(* CoDeSys 2.3.9.48 project: 20170913_WUR_added_Inverter_Control.pro *)
(* Version: 0.9 *)
(* Description: Project Distributie Automatisering *)
(* Libraries: Serial_Interface_01.lib 22.4.13 12:50:14, Util.lib 30.1.13 13:05:12, WagoLib787_01.lib 10.11.14 13:02:32, mod_com.lib 30.1.13 13:05:12, WagoConfigToolLIB.lib 30.1.13 13:05:12, PowerMeasurement_495_02.lib 13.9.17 08:23:51, SysLibTime.lib 30.1.13 13:05:12, WagoLibSHA1.lib 19.8.11 14:53:16, WagoLibMySQL_03.lib 23.7.14 09:13:36, SerComm.lib 30.1.13 13:05:12, SysLibSockets.lib 22.5.14 16:16:32, SysLibFile.lib 30.1.13 13:05:12, SysLibMem.lib 30.1.13 13:05:12, SysLibSem.lib 30.1.13 13:05:12, SysLibRtc.lib 30.1.13 13:05:12, WagoLibEthernet_01.lib 1.4.15 14:24:28, WAGOLIBNTP.lib 19.8.11 14:53:14, Modb_l05.lib 13.5.15 10:30:08, SysLibDir.lib 30.1.13 13:05:12, C:\Program Files\WAGO Software\CODESYS V2.3\Targets\WAGO\Libraries\32_Bit\WAGO_Datalogger_02.lib 5.4.17 15:41:49, Wago_MBCFG_SERIAL_01.lib 1.4.15 14:24:28, Wago_MBCFG_COMMON_01.lib 1.4.15 14:24:28, Standard.lib 20.5.14 08:13:26, Iecsfc.lib 30.1.13 13:05:12, SYSLIBCALLBACK.LIB 30.1.13 13:05:12 *)

(* PLC configuration (modules and I/O channels)
0750-0430 8 DI 24 V DC 3.0ms [Type_1_8_Channels] node 0, in %IB264 out %QB280
  AT %IX132.0 [BOOLOnX_I] Ch_1 Digital input
  AT %IX132.1 [BOOLOnX_I] Ch_2 Digital input
  AT %IX132.2 [BOOLOnX_I] Ch_3 Digital input
  AT %IX132.3 [BOOLOnX_I] Ch_4 Digital input
  AT %IX132.4 [BOOLOnX_I] Ch_5 Digital input
  AT %IX132.5 [BOOLOnX_I] Ch_6 Digital input
  AT %IX132.6 [BOOLOnX_I] Ch_7 Digital input
  AT %IX132.7 [BOOLOnX_I] Ch_8 Digital input
0750-0430 8 DI 24 V DC 3.0ms [Type_1_8_Channels] node 1, in %IB264 out %QB280
  AT %IX132.8 [BOOLOnX_I] Ch_1 Digital input
  AT %IX132.9 [BOOLOnX_I] Ch_2 Digital input
  AT %IX132.10 [BOOLOnX_I] Ch_3 Digital input
  AT %IX132.11 [BOOLOnX_I] Ch_4 Digital input
  AT %IX132.12 [BOOLOnX_I] Ch_5 Digital input
  AT %IX132.13 [BOOLOnX_I] Ch_6 Digital input
  AT %IX132.14 [BOOLOnX_I] Ch_7 Digital input
  AT %IX132.15 [BOOLOnX_I] Ch_8 Digital input
0750-0430 8 DI 24 V DC 3.0ms [Type_1_8_Channels] node 2, in %IB265 out %QB280
  AT %IX133.0 [BOOLOnX_I] Ch_1 Digital input
  AT %IX133.1 [BOOLOnX_I] Ch_2 Digital input
  AT %IX133.2 [BOOLOnX_I] Ch_3 Digital input
  AT %IX133.3 [BOOLOnX_I] Ch_4 Digital input
  AT %IX133.4 [BOOLOnX_I] Ch_5 Digital input
  AT %IX133.5 [BOOLOnX_I] Ch_6 Digital input
  AT %IX133.6 [BOOLOnX_I] Ch_7 Digital input
  AT %IX133.7 [BOOLOnX_I] Ch_8 Digital input
0750-0430 8 DI 24 V DC 3.0ms [Type_1_8_Channels] node 3, in %IB266 out %QB280
  AT %IX133.8 [BOOLOnX_I] Ch_1 Digital input
  AT %IX133.9 [BOOLOnX_I] Ch_2 Digital input
  AT %IX133.10 [BOOLOnX_I] Ch_3 Digital input
  AT %IX133.11 [BOOLOnX_I] Ch_4 Digital input
  AT %IX133.12 [BOOLOnX_I] Ch_5 Digital input
  AT %IX133.13 [BOOLOnX_I] Ch_6 Digital input
  AT %IX133.14 [BOOLOnX_I] Ch_7 Digital input
  AT %IX133.15 [BOOLOnX_I] Ch_8 Digital input
0750-0430 8 DI 24 V DC 3.0ms [Type_1_8_Channels] node 4, in %IB267 out %QB280
  AT %IX134.0 [BOOLOnX_I] Ch_1 Digital input
  AT %IX134.1 [BOOLOnX_I] Ch_2 Digital input
  AT %IX134.2 [BOOLOnX_I] Ch_3 Digital input
  AT %IX134.3 [BOOLOnX_I] Ch_4 Digital input
  AT %IX134.4 [BOOLOnX_I] Ch_5 Digital input
  AT %IX134.5 [BOOLOnX_I] Ch_6 Digital input
  AT %IX134.6 [BOOLOnX_I] Ch_7 Digital input
  AT %IX134.7 [BOOLOnX_I] Ch_8 Digital input
0750-0530 8 DO 24 V DC 0.5A [Type_10_8_Channels] node 5, in %IB268 out %QB280
  AT %QX140.0 [BOOLOnX_Q] Ch_1 Digital output
  AT %QX140.1 [BOOLOnX_Q] Ch_2 Digital output
  AT %QX140.2 [BOOLOnX_Q] Ch_3 Digital output
  AT %QX140.3 [BOOLOnX_Q] Ch_4 Digital output
  AT %QX140.4 [BOOLOnX_Q] Ch_5 Digital output
  AT %QX140.5 [BOOLOnX_Q] Ch_6 Digital output
  AT %QX140.6 [BOOLOnX_Q] Ch_7 Digital output
  AT %QX140.7 [BOOLOnX_Q] Ch_8 Digital output
0750-0530 8 DO 24 V DC 0.5A [Type_10_8_Channels] node 6, in %IB269 out %QB280
  AT %QX140.8 [BOOLOnX_Q] Ch_1 Digital output
  AT %QX140.9 [BOOLOnX_Q] Ch_2 Digital output
  AT %QX140.10 [BOOLOnX_Q] Ch_3 Digital output
  AT %QX140.11 [BOOLOnX_Q] Ch_4 Digital output
  AT %QX140.12 [BOOLOnX_Q] Ch_5 Digital output
  AT %QX140.13 [BOOLOnX_Q] Ch_6 Digital output
  AT %QX140.14 [BOOLOnX_Q] Ch_7 Digital output
  AT %QX140.15 [BOOLOnX_Q] Ch_8 Digital output
0750-0530 8 DO 24 V DC 0.5A [Type_10_8_Channels] node 7, in %IB269 out %QB281
  AT %QX141.0 [BOOLOnX_Q] Ch_1 Digital output
  AT %QX141.1 [BOOLOnX_Q] Ch_2 Digital output
  AT %QX141.2 [BOOLOnX_Q] Ch_3 Digital output
  AT %QX141.3 [BOOLOnX_Q] Ch_4 Digital output
  AT %QX141.4 [BOOLOnX_Q] Ch_5 Digital output
  AT %QX141.5 [BOOLOnX_Q] Ch_6 Digital output
  AT %QX141.6 [BOOLOnX_Q] Ch_7 Digital output
  AT %QX141.7 [BOOLOnX_Q] Ch_8 Digital output
0750-0530 8 DO 24 V DC 0.5A [Type_10_8_Channels] node 8, in %IB269 out %QB282
  AT %QX141.8 [BOOLOnX_Q] Ch_1 Digital output
  AT %QX141.9 [BOOLOnX_Q] Ch_2 Digital output
  AT %QX141.10 [BOOLOnX_Q] Ch_3 Digital output
  AT %QX141.11 [BOOLOnX_Q] Ch_4 Digital output
  AT %QX141.12 [BOOLOnX_Q] Ch_5 Digital output
  AT %QX141.13 [BOOLOnX_Q] Ch_6 Digital output
  AT %QX141.14 [BOOLOnX_Q] Ch_7 Digital output
  AT %QX141.15 [BOOLOnX_Q] Ch_8 Digital output
AT %QW0 [WORDOnW_Q] Ch_1 Analog output
AT %QW1 [WORDOnW_Q] Ch_2 Analog output
AT %QW2 [WORDOnW_Q] Ch_3 Analog output
AT %QW3 [WORDOnW_Q] Ch_4 Analog output
AT %QW4 [WORDOnW_Q] Ch_1 Analog output
AT %QW5 [WORDOnW_Q] Ch_2 Analog output
AT %QW6 [WORDOnW_Q] Ch_3 Analog output
AT %QW7 [WORDOnW_Q] Ch_4 Analog output
0750-0495/0000-0001 3-phase PoM690/ 5A [Type_58_1_Channels] node 11, in %IB240 out %QB264
  AT %IW0 [WORDOnW_I] Status Word
  AT %IW1 [WORDOnW_I] Status Word 1
  AT %IW2 [WORDOnW_I] Status Word 2
  AT %IW3 [WORDOnW_I] Status Word 3
  AT %ID2 [DWORDOnD_I] process value 1
  AT %ID3 [DWORDOnD_I] process value 2
  AT %ID4 [DWORDOnD_I] process value 3
  AT %ID5 [DWORDOnD_I] process value 4
  AT %QW8 [WORDOnW_Q] Control Word
  AT %QW9 [WORDOnW_Q] Control Word 1
  AT %QW10 [WORDOnW_Q] Control Word 2
  AT %QW11 [WORDOnW_Q] Control Word 3
0750-0495/0000-0001 3-phase PoM690/ 5A [Type_58_1_Channels] node 12, in %IB240 out %QB272
  AT %IW12 [WORDOnW_I] Status Word
  AT %IW13 [WORDOnW_I] Status Word 1
  AT %IW14 [WORDOnW_I] Status Word 2
  AT %IW15 [WORDOnW_I] Status Word 3
  AT %ID8 [DWORDOnD_I] process value 1
  AT %ID9 [DWORDOnD_I] process value 2
  AT %ID10 [DWORDOnD_I] process value 3
  AT %ID11 [DWORDOnD_I] process value 4
  AT %QW20 [WORDOnW_Q] Control Word
  AT %QW21 [WORDOnW_Q] Control Word 1
  AT %QW22 [WORDOnW_Q] Control Word 2
  AT %QW23 [WORDOnW_Q] Control Word 3
0750-0495/0000-0001 3-phase PoM690/ 5A [Type_58_1_Channels] node 13, in %IB264 out %QB296
  AT %IW24 [WORDOnW_I] Status Word
  AT %IW25 [WORDOnW_I] Status Word 1
  AT %IW26 [WORDOnW_I] Status Word 2
  AT %IW27 [WORDOnW_I] Status Word 3
  AT %ID14 [DWORDOnD_I] process value 1
  AT %ID15 [DWORDOnD_I] process value 2
  AT %ID16 [DWORDOnD_I] process value 3
  AT %ID17 [DWORDOnD_I] process value 4
  AT %QW32 [WORDOnW_Q] Control Word
  AT %QW33 [WORDOnW_Q] Control Word 1
  AT %QW34 [WORDOnW_Q] Control Word 2
  AT %QW35 [WORDOnW_Q] Control Word 3
0750-0495/0000-0001 3-phase PoM690/ 5A [Type_58_1_Channels] node 14, in %IB288 out %QB320
  AT %IW36 [WORDOnW_I] Status Word
  AT %IW37 [WORDOnW_I] Status Word 1
  AT %IW38 [WORDOnW_I] Status Word 2
  AT %IW39 [WORDOnW_I] Status Word 3
  AT %ID20 [DWORDOnD_I] process value 1
  AT %ID21 [DWORDOnD_I] process value 2
  AT %ID22 [DWORDOnD_I] process value 3
  AT %ID23 [DWORDOnD_I] process value 4
  AT %QW44 [WORDOnW_Q] Control Word
  AT %QW45 [WORDOnW_Q] Control Word 1
  AT %QW46 [WORDOnW_Q] Control Word 2
  AT %QW47 [WORDOnW_Q] Control Word 3
0750-0495/0000-0001 3-phase PoM690/ 5A [Type_58_1_Channels] node 15, in %IB312 out %QB344
  AT %IW48 [WORDOnW_I] Status Word
  AT %IW49 [WORDOnW_I] Status Word 1
  AT %IW50 [WORDOnW_I] Status Word 2
  AT %IW51 [WORDOnW_I] Status Word 3
  AT %ID26 [DWORDOnD_I] process value 1
  AT %ID27 [DWORDOnD_I] process value 2
  AT %ID28 [DWORDOnD_I] process value 3
  AT %ID29 [DWORDOnD_I] process value 4
  AT %QW56 [WORDOnW_Q] Control Word
  AT %QW57 [WORDOnW_Q] Control Word 1
  AT %QW58 [WORDOnW_Q] Control Word 2
  AT %QW59 [WORDOnW_Q] Control Word 3
0750-0495/0000-0001 3-phase PoM690/ 5A [Type_58_1_Channels] node 16, in %IB336 out %QB368
  AT %IW60 [WORDOnW_I] Status Word
  AT %IW61 [WORDOnW_I] Status Word 1
  AT %IW62 [WORDOnW_I] Status Word 2
  AT %IW63 [WORDOnW_I] Status Word 3
  AT %ID32 [DWORDOnD_I] process value 1
  AT %ID33 [DWORDOnD_I] process value 2
  AT %ID34 [DWORDOnD_I] process value 3
  AT %ID35 [DWORDOnD_I] process value 4
  AT %QW68 [WORDOnW_Q] Control Word
  AT %QW69 [WORDOnW_Q] Control Word 1
  AT %QW70 [WORDOnW_Q] Control Word 2
  AT %QW71 [WORDOnW_Q] Control Word 3
0750-0495/0000-0001 3-phase PoM690/ 5A [Type_58_1_Channels] node 17, in %IB360 out %QB392
  AT %IW72 [WORDOnW_I] Status Word
  AT %IW73 [WORDOnW_I] Status Word 1
  AT %IW74 [WORDOnW_I] Status Word 2
  AT %IW75 [WORDOnW_I] Status Word 3
  AT %ID38 [DWORDOnD_I] process value 1
  AT %ID39 [DWORDOnD_I] process value 2
  AT %ID40 [DWORDOnD_I] process value 3
  AT %ID41 [DWORDOnD_I] process value 4
  AT %QW80 [WORDOnW_Q] Control Word
  AT %QW81 [WORDOnW_Q] Control Word 1
  AT %QW82 [WORDOnW_Q] Control Word 2
  AT %QW83 [WORDOnW_Q] Control Word 3
0750-0495/0000-0001 3-phase PoM690/ 5A [Type_58_1_Channels] node 18, in %IB384 out %QB416
  AT %IW84 [WORDOnW_I] Status Word
  AT %IW85 [WORDOnW_I] Status Word 1
  AT %IW86 [WORDOnW_I] Status Word 2
  AT %IW87 [WORDOnW_I] Status Word 3
  AT %ID44 [DWORDOnD_I] process value 1
  AT %ID45 [DWORDOnD_I] process value 2
  AT %ID46 [DWORDOnD_I] process value 3
  AT %ID47 [DWORDOnD_I] process value 4
  AT %QW92 [WORDOnW_Q] Control Word
  AT %QW93 [WORDOnW_Q] Control Word 1
  AT %QW94 [WORDOnW_Q] Control Word 2
  AT %QW95 [WORDOnW_Q] Control Word 3
0750-0495/0000-0001 3-phase PoM690/ 5A [Type_58_1_Channels] node 19, in %IB408 out %QB440
  AT %IW96 [WORDOnW_I] Status Word
  AT %IW97 [WORDOnW_I] Status Word 1
  AT %IW98 [WORDOnW_I] Status Word 2
  AT %IW99 [WORDOnW_I] Status Word 3
  AT %ID50 [DWORDOnD_I] process value 1
  AT %ID51 [DWORDOnD_I] process value 2
  AT %ID52 [DWORDOnD_I] process value 3
  AT %ID53 [DWORDOnD_I] process value 4
  AT %QW104 [WORDOnW_Q] Control Word
  AT %QW105 [WORDOnW_Q] Control Word 1
  AT %QW106 [WORDOnW_Q] Control Word 2
  AT %QW107 [WORDOnW_Q] Control Word 3
0750-0495/0000-0001 3-phase PoM690/ 5A [Type_58_1_Channels] node 20, in %IB432 out %QB464
  AT %IW108 [WORDOnW_I] Status Word
  AT %IW109 [WORDOnW_I] Status Word 1
  AT %IW110 [WORDOnW_I] Status Word 2
  AT %IW111 [WORDOnW_I] Status Word 3
  AT %ID56 [DWORDOnD_I] process value 1
  AT %ID57 [DWORDOnD_I] process value 2
  AT %ID58 [DWORDOnD_I] process value 3
  AT %ID59 [DWORDOnD_I] process value 4
  AT %QW116 [WORDOnW_Q] Control Word
  AT %QW117 [WORDOnW_Q] Control Word 1
  AT %QW118 [WORDOnW_Q] Control Word 2
  AT %QW119 [WORDOnW_Q] Control Word 3
0750-0495/0000-0001 3-phase PoM690/ 5A [Type_58_1_Channels] node 0, in %IB456 out %QB488
  AT %IW120 [WORDOnW_I] Status Word
  AT %IW121 [WORDOnW_I] Status Word 1
  AT %IW122 [WORDOnW_I] Status Word 2
  AT %IW123 [WORDOnW_I] Status Word 3
  AT %ID62 [DWORDOnD_I] process value 1
  AT %ID63 [DWORDOnD_I] process value 2
  AT %ID64 [DWORDOnD_I] process value 3
  AT %ID65 [DWORDOnD_I] process value 4
  AT %QW128 [WORDOnW_Q] Control Word
  AT %QW129 [WORDOnW_Q] Control Word 1
  AT %QW130 [WORDOnW_Q] Control Word 2
  AT %QW131 [WORDOnW_Q] Control Word 3
REAL, Fieldbus output [MODBUS_REAL_OUT] node 0, in %IB0 out %QB0
  mb_var0 AT %QD500 [REALOnD_Q] TEST
Modbus-Master [MB_MASTER] node 2, in %IB0 out %QB0
*)

(* Task configuration *)
TASK Test (PRIORITY := 2); (* freewheeling *)
	variables_to_system_array();
	SynchroniserSwitch();
	Group2();
END_TASK
TASK WriteData (PRIORITY := 31, INTERVAL := T#1000ms);
	WRITE_DATA();
END_TASK
TASK Switching (PRIORITY := 3); (* freewheeling *)
	Group1();
END_TASK
TASK Measurements (PRIORITY := 1); (* freewheeling *)
	run_PQ();
END_TASK
TASK Control (PRIORITY := 0, INTERVAL := T#1000ms);
	CHP_Controller();
	EV_Controller();
	Mixer_Controller();
	Inverter_Control_1();
	Inverter_Control_2();
END_TASK

(* Global variable list: Global_Variables *)
VAR_GLOBAL
(* testing purpose values *)
	x																:	 REAL:=1;

(* internally used variables *)
	r_Battery_Bus_Frequency									:	 REAL;
	r_Battery_Bus_Voltage										:	 REAL;
	r_Grid_Bus_Frequency										:	 REAL;
	r_Grid_Bus_Voltage											:	 REAL;

(* Array containing all the system parameters. Values are accessable through modbus tcp starting from register 12288. REAL uses two registers per variable *)
	arSystemState									AT %MW0	:	ARRAY[0.. iNumberSystemVar] OF REAL;
	arSystemStateNames										:	ARRAY[0.. iNumberSystemVar] OF STRING; (* names of registers used in mysql write *)

 (*Measurement values for cards*)
	arMeasurementsGroup1							:	ARRAY[1.. iNumberMeasurementVar] OF REAL;
	arMeasurementsGroup2							:	ARRAY[1.. iNumberMeasurementVar] OF REAL;
	arMeasurementsGroup3							:	ARRAY[1.. iNumberMeasurementVar] OF REAL;
	arMeasurementsGroup4							:	ARRAY[1.. iNumberMeasurementVar] OF REAL;
	arMeasurementsGroup5							:	ARRAY[1.. iNumberMeasurementVar] OF REAL;
	arMeasurementsGroup6							:	ARRAY[1.. iNumberMeasurementVar] OF REAL;
	arMeasurementsGroup7							:	ARRAY[1.. iNumberMeasurementVar] OF REAL;
	arMeasurementsGroup8							:	ARRAY[1.. iNumberMeasurementVar] OF REAL;
	arMeasurementsGroup9							:	ARRAY[1.. iNumberMeasurementVar] OF REAL;
	arMeasurementsGroupA							:	ARRAY[1.. iNumberMeasurementVar] OF REAL;
	arMeasurementsGroupB							:	ARRAY[1.. iNumberMeasurementVar] OF REAL;

 (*Measurement values for bus connector from janitza*)
(* ___ OLD____
	r_modbus_Bus_Connector_L1_P				:  REAL;
	r_modbus_Bus_Connector_L2_P				:  REAL;
	r_modbus_Bus_Connector_L3_P				:  REAL;
	r_modbus_Bus_Connector_L1_Q				:  REAL;
	r_modbus_Bus_Connector_L2_Q				:  REAL;
	r_modbus_Bus_Connector_L3_Q				:  REAL;
	r_modbus_Bus_Connector_L1_V				:  REAL;
	r_modbus_Bus_Connector_L2_V				:  REAL;
	r_modbus_Bus_Connector_L3_V				:  REAL;
	r_modbus_Bus_Connector_L1_I				:  REAL;
	r_modbus_Bus_Connector_L2_I				:  REAL;
	r_modbus_Bus_Connector_L3_I				:  REAL;
	r_modbus_Bus_Connector_L1_f				:  REAL;
	r_modbus_Bus_Connector_L2_f				:  REAL;
	r_modbus_Bus_Connector_L3_f				:  REAL;
*)
	Bus_Connector_L1_P : REAL;
	Bus_Connector_L2_P : REAL;
	Bus_Connector_L3_P : REAL;
	Bus_Connector_L1_Q : REAL;
	Bus_Connector_L2_Q : REAL;
	Bus_Connector_L3_Q : REAL;
	Bus_Connector_L1_V : REAL;
	Bus_Connector_L2_V : REAL;
	Bus_Connector_L3_V : REAL;
	Bus_Connector_L1_I : REAL;
	Bus_Connector_L2_I : REAL;
	Bus_Connector_L3_I : REAL;
	Bus_Connector_L1_f : REAL;
	Bus_Connector_L2_f : REAL;
	Bus_Connector_L3_f : REAL;
	Bus_Connector_3F_radians : REAL;

(* DEIF SYNCHRONISER SWITCHING VARIABLES (including variable set from modbus object < doesnt exist jet *)
(* ___OLD ___
	r_modbus_Synchroniser_state					:	REAL:= 1; (* 0 = deny, 1 = allow, 2 = close request*)
	r_modbus_Synchroniser_Denied_Request		:	BOOL;
	r_modbus_Synchroniser_Close_Request		:	BOOL;

	r_DI_Synchroniser_Close_Request				:	BOOL;
	r_DI_Synchroniser_Denied_Request			:	BOOL;
	r_DI_Synchroniser_Closed						:	BOOL;

	r_Synchroniser_Close_Request_Relais		:	BOOL;
	r_Synchroniser_Close_Denied_Relais			:	BOOL; (* only inplemented if hardware output is available (to control panelel LED*)
*)

	Bus_Connector_3F_Sync_close_requested   			AT %QX129.2 : BOOL;
	Bus_Connector_3F_Sync_closed   						AT %IX121.12 : BOOL;
	Bus_Connector_3F_Sync_close_requested_panel    	AT %IX121.13 : BOOL;
	Bus_Connector_3F_Sync_denied_panel   				AT %IX121.14 : BOOL;
	Bus_Connector_3F_Sync_close_requested_modbus 					: BOOL;
	Bus_Connector_3F_Sync_denied_modbus				 				: BOOL;
	Bus_Connector_3F_Field_Rotation										: REAL;
	r_Synchroniser_Close_Denied_Relais (* ?LED? *)						: BOOL;


(* Group Switching states ______ OLD__________
	Group1_autoswitch_state 						(*AT %IX0.0*)	:	BOOL;
	Group1_gridbus_switch_state 					(*AT %QX0.0*)	:	BOOL;
	Group1_batterybus_switch_state 				(*AT %QX0.0*)	:	BOOL;
	Group2_autoswitch_state 						(*AT %IX0.0*)	:	BOOL;
	Group2_gridbus_switch_state 					(*AT %QX0.0*)	:	BOOL;
	Group2_batterybus_switch_state 				(*AT %QX0.0*)	:	BOOL;
	Group3_autoswitch_state 						(*AT %IX0.0*)	:	BOOL;
	Group3_gridbus_switch_state 					(*AT %QX0.0*)	:	BOOL;
	Group3_batterybus_switch_state 				(*AT %QX0.0*)	:	BOOL;
	Group4_autoswitch_state 						(*AT %IX0.0*)	:	BOOL;
	Group4_gridbus_switch_state 					(*AT %QX0.0*)	:	BOOL;
	Group4_batterybus_switch_state 				(*AT %QX0.0*)	:	BOOL;
	Group5_autoswitch_state 						(*AT %IX0.0*)	:	BOOL;
	Group5_gridbus_switch_state 					(*AT %QX0.0*)	:	BOOL;
	Group5_batterybus_switch_state 				(*AT %QX0.0*)	:	BOOL;
	Group6_autoswitch_state 						(*AT %IX0.0*)	:	BOOL;
	Group6_gridbus_switch_state 					(*AT %QX0.0*)	:	BOOL;
	Group6_batterybus_switch_state 				(*AT %QX0.0*)	:	BOOL;
	Group7_autoswitch_state 						(*AT %IX0.0*)	:	BOOL;
	Group7_gridbus_switch_state 					(*AT %QX0.0*)	:	BOOL;
	Group7_batterybus_switch_state 				(*AT %QX0.0*)	:	BOOL;
	Group8_autoswitch_state 						(*AT %IX0.0*)	:	BOOL;
	Group8_gridbus_switch_state 					(*AT %QX0.0*)	:	BOOL;
	Group8_batterybus_switch_state 				(*AT %QX0.0*)	:	BOOL;
	Group9_autoswitch_state 						(*AT %IX0.0*)	:	BOOL;
	Group9_gridbus_switch_state 					(*AT %QX0.0*)	:	BOOL;
	Group9_batterybus_switch_state 				(*AT %QX0.0*)	:	BOOL;
	Group10_autoswitch_state 						(*AT %IX0.0*)	:	BOOL;
	Group10_gridbus_switch_state 					(*AT %QX0.0*)	:	BOOL;
	Group10_batterybus_switch_state 				(*AT %QX0.0*)	:	BOOL;
	Group11_autoswitch_state 						(*AT %IX0.0*)	:	BOOL;
	Group11_gridbus_switch_state 					(*AT %QX0.0*)	:	BOOL;
	Group11_batterybus_switch_state 				(*AT %QX0.0*)	:	BOOL;
*)

	Group_control_Frequencybased_bus_selecting_state : REAL:=0;
	Group_control_min_time_above_switch_frequency : REAL := 2000;
	Group_control_min_time_below_switch_frequency : REAL := 2000;
	Group1_3F_Switch_frequency_to_batterybus : REAL;
	Group1_3F_Switch_frequency_to_gridbus : REAL;
	Group1_3F_min_time_between_switching : REAL:= 10000;
	Group2_3F_Switch_frequency_to_batterybus : REAL := 51;
	Group2_3F_Switch_frequency_to_gridbus : REAL := 49;
	Group2_3F_min_time_between_switching : REAL := 10000;
	Group3_3F_Switch_frequency_to_batterybus : REAL;
	Group3_3F_Switch_frequency_to_gridbus : REAL;
	Group3_3F_min_time_between_switching : REAL;
	Group4_3F_Switch_frequency_to_batterybus : REAL;
	Group4_3F_Switch_frequency_to_gridbus : REAL;
	Group4_3F_min_time_between_switching : REAL;
	Group5_3F_Switch_frequency_to_batterybus : REAL;
	Group5_3F_Switch_frequency_to_gridbus : REAL;
	Group5_3F_min_time_between_switching : REAL;
	Group6_3F_Switch_frequency_to_batterybus : REAL;
	Group6_3F_Switch_frequency_to_gridbus : REAL;
	Group6_3F_min_time_between_switching : REAL;
	Group7_3F_Switch_frequency_to_batterybus : REAL;
	Group7_3F_Switch_frequency_to_gridbus : REAL;
	Group7_3F_min_time_between_switching : REAL;
	Group8_3F_Switch_frequency_to_batterybus : REAL;
	Group8_3F_Switch_frequency_to_gridbus : REAL;
	Group8_3F_min_time_between_switching : REAL;
	Group9_3F_Switch_frequency_to_batterybus : REAL;
	Group9_3F_Switch_frequency_to_gridbus : REAL;
	Group9_3F_min_time_between_switching : REAL;

(* frequency based swithcing parameters *)
	Frequencybased_bus_selecting_state							:  BOOL	:= FALSE;
	Switch_Gap_Time												:  INT		:= 2000;
(*
	Group1_Switch_frequency_to_batterybus						:  REAL	 := 52;
	Group1_Switch_frequency_to_gridbus							:  REAL	 := 48;
	Group1_min_time_above_switch_frequency					:  INT 		:= 10000; (*ms*)
	Group1_min_time_below_switch_frequency					:  INT 		:= 10000; (*ms*)
	Group1_min_time_between_switching							:  INT 		:= 10000; (*ms*)
	Group2_Switch_frequency_to_batterybus						:  REAL 	:= 52;
	Group2_Switch_frequency_to_gridbus							:  REAL 	:= 48;
	Group2_min_time_above_switch_frequency					:  INT 		:= 10000; (*ms*)
	Group2_min_time_below_switch_frequency					:  INT 		:= 10000; (*ms*)
	Group2_min_time_between_switching							:  INT 		:= 10000; (*ms*)
	Group3_Switch_frequency_to_batterybus						:  REAL 	:= 52;
	Group3_Switch_frequency_to_gridbus							:  REAL 	:= 48;
	Group3_min_time_above_switch_frequency					:  INT 		:= 10000; (*ms*)
	Group3_min_time_below_switch_frequency					:  INT 		:= 10000; (*ms*)
	Group3_min_time_between_switching							:  INT 		:= 10000; (*ms*)
	Group4_Switch_frequency_to_batterybus						:  REAL 	:= 52;
	Group4_Switch_frequency_to_gridbus							:  REAL 	:= 48;
	Group4_min_time_above_switch_frequency					:  INT 		:= 10000; (*ms*)
	Group4_min_time_below_switch_frequency					:  INT 		:= 10000; (*ms*)
	Group4_min_time_between_switching							:  INT 		:= 10000; (*ms*)
	Group5_Switch_frequency_to_batterybus						:  REAL 	:= 52;
	Group5_Switch_frequency_to_gridbus							:  REAL 	:= 48;
	Group5_min_time_above_switch_frequency					:  INT 		:= 10000; (*ms*)
	Group5_min_time_below_switch_frequency					:  INT 		:= 10000; (*ms*)
	Group5_min_time_between_switching							:  INT 		:= 10000; (*ms*)
	Group6_Switch_frequency_to_batterybus						:  REAL 	:= 52;
	Group6_Switch_frequency_to_gridbus							:  REAL 	:= 48;
	Group6_min_time_above_switch_frequency					:  INT 		:= 10000; (*ms*)
	Group6_min_time_below_switch_frequency					:  INT 		:= 10000; (*ms*)
	Group6_min_time_between_switching							:  INT 		:= 10000; (*ms*)
	Group7_Switch_frequency_to_batterybus						:  REAL 	:= 52;
	Group7_Switch_frequency_to_gridbus							:  REAL 	:= 48;
	Group7_min_time_above_switch_frequency					:  INT 		:= 10000; (*ms*)
	Group7_min_time_below_switch_frequency					:  INT 		:= 10000; (*ms*)
	Group7_min_time_between_switching							:  INT 		:= 10000; (*ms*)
	Group8_Switch_frequency_to_batterybus						:  REAL 	:= 52;
	Group8_Switch_frequency_to_gridbus							:  REAL 	:= 48;
	Group8_min_time_above_switch_frequency					:  INT 		:= 10000; (*ms*)
	Group8_min_time_below_switch_frequency					:  INT 		:= 10000; (*ms*)
	Group8_min_time_between_switching							:  INT 		:= 10000; (*ms*)
	Group9_Switch_frequency_to_batterybus						:  REAL 	:= 52;
	Group9_Switch_frequency_to_gridbus							:  REAL 	:= 48;
	Group9_min_time_above_switch_frequency					:  INT 		:= 10000; (*ms*)
	Group9_min_time_below_switch_frequency					:  INT 		:= 10000; (*ms*)
	Group9_min_time_between_switching							:  INT 		:= 10000; (*ms*)
*)

	CHP_control_grid_bus_select_controlswitch 							: BOOL;
	CHP_control_baterry_bus_select_controlswitch 						: BOOL;
	CHP_control_auto_bus_select_controlswitch 							: BOOL;
	CHP_control_Offgrid_request    							AT %QX129.4  : BOOL;
	CHP_control_internal_contacter_switch_state  			AT %IX121.15 : BOOL;
	CHP_gridbus_switch_state												: BOOL; (*request from battery bus frequency *)
	CHP_batterybus_switch_state											: BOOL; (*request from battery bus frequency *)

	Inverter_10V_control_Max_Freq_Ref							:  INT		:= 51;  (* Maximum freq possible on the battery bus or te highest freq you want to scale the 0-10V analog output to*)
	Inverter_10V_control_Min_Freq_Ref							:  INT		:= 49;  (* Minimum freq possible on the battery bus or te loweste freq you want to scale the 0-10V analog output to*)
(* Analog Out Controller variables *)

	Mixer_control_control_signal 							AT %QW0 : REAL;   (*0-10V*)
	EV_control_control_signal   								AT %QW2 : REAL;   (*0-10V *)
	CHP_control_Offgrid_Active_Power_control				AT %QW4 : REAL;   (* 4-20ma *)
	Inverter_control1_signal   								AT %QW1 : REAL;	  (*0-10V*)
	Inverter_control2_signal									AT %QW3 : REAL;	  (*0-10V*)
	Group1_3F_Auto_relay_control_battery_bus   	AT %QX128.1  : BOOL;
	Group1_3F_Auto_relay_control_grid_bus   		AT %QX128.0  : BOOL;
	Group1_3F_Selector_auto_bus_select    		AT %IX121.2 : BOOL;
	Group1_3F_relay_state_battery_bus   			AT %IX120.1  : BOOL;
	Group1_3F_relay_state_grid_bus   				AT %IX120.0  : BOOL;
	Group2_3F_Auto_relay_control_battery_bus   	AT %QX128.3  : BOOL;
	Group2_3F_Auto_relay_control_grid_bus   		AT %QX128.2  : BOOL;
	Group2_3F_Selector_auto_bus_select  			AT %IX121.3 : BOOL;
	Group2_3F_relay_state_battery_bus   			AT %IX120.3  : BOOL;
	Group2_3F_relay_state_grid_bus   				AT %IX120.2  : BOOL;
	Group3_3F_Auto_relay_control_battery_bus   	AT %QX128.5  : BOOL;
	Group3_3F_Auto_relay_control_grid_bus   		AT %QX128.4  : BOOL;
	Group3_3F_Selector_auto_bus_select   		AT %IX121.4 : BOOL;
	Group3_3F_relay_state_battery_bus   			AT %IX120.5  : BOOL;
	Group3_3F_relay_state_grid_bus   				AT %IX120.4  : BOOL;
	Group4_3F_Auto_relay_control_battery_bus    	AT %QX128.7  : BOOL;
	Group4_3F_Auto_relay_control_grid_bus    		AT %QX128.6  : BOOL;
	Group4_3F_Selector_auto_bus_select   		AT %IX121.5 : BOOL;
	Group4_3F_relay_state_battery_bus   			AT %IX120.7  : BOOL;
	Group4_3F_relay_state_grid_bus   				AT %IX120.6  : BOOL;
	Group5_3F_Auto_relay_control_battery_bus   	AT %QX128.9  : BOOL;
	Group5_3F_Auto_relay_control_grid_bus   		AT %QX128.8  : BOOL;
	Group5_3F_Selector_auto_bus_select   		AT %IX121.6 : BOOL;
	Group5_3F_relay_state_battery_bus   			AT %IX120.9  : BOOL;
	Group5_3F_relay_state_grid_bus   				AT %IX120.8  : BOOL;
	Group6_3F_Auto_relay_control_battery_bus   	AT %QX128.11  : BOOL;
	Group6_3F_Auto_relay_control_grid_bus   		AT %QX128.10  : BOOL;
	Group6_3F_Selector_auto_bus_select   		AT %IX121.7 : BOOL;
	Group6_3F_relay_state_battery_bus   			AT %IX120.11  : BOOL;
	Group6_3F_relay_state_grid_bus   				AT %IX120.10  : BOOL;
	Group7_3F_Auto_relay_control_battery_bus   	AT %QX128.13  : BOOL;
	Group7_3F_Auto_relay_control_grid_bus   		AT %QX128.12  : BOOL;
	Group7_3F_Selector_auto_bus_select   		AT %IX121.8 : BOOL;
	Group7_3F_relay_state_battery_bus   			AT %IX120.13  : BOOL;
	Group7_3F_relay_state_grid_bus   				AT %IX120.12  : BOOL;
	Group8_3F_Auto_relay_control_battery_bus   	AT %QX128.15  : BOOL;
	Group8_3F_Auto_relay_control_grid_bus   		AT %QX128.14  : BOOL;
	Group8_3F_Selector_auto_bus_select   		AT %IX121.9 : BOOL;
	Group8_3F_relay_state_battery_bus   			AT %IX120.15  : BOOL;
	Group8_3F_relay_state_grid_bus   				AT %IX120.14  : BOOL;
	Group9_3F_Auto_relay_control_battery_bus   	AT %QX129.1  : BOOL;
	Group9_3F_Auto_relay_control_grid_bus   		AT %QX129.0  : BOOL;
	Group9_3F_Selector_auto_bus_select   		AT %IX121.10 : BOOL;
	Group9_3F_relay_state_battery_bus   			AT %IX121.1  : BOOL;
	Group9_3F_relay_state_grid_bus   				AT %IX121.0  : BOOL;

(* Controm panel LEDs *)
	Control_panel_status_warning_led   			AT %QX129.12  : BOOL;
	Control_panel_status_error_led   				AT %QX129.13  : BOOL;
	Control_panel_status_operational_led    		AT %QX129.11  : BOOL;

END_VAR

VAR_GLOBAL CONSTANT

(* Read / write CSV-files *)
	iMaxParams			:	INT:=8;(* Number of Parameters per File *)
	gc_ParameterCount	:	INT:=1;(* Number of Values per Parameter *)
	gc_RawDataSize		:	UINT:=500; (* Raw data size for reading in file ASCII *)
	gcRowExcel			:	INT:=1;

(* meaasurement array length *)
	iNumberMeasurementVar		:	INT := 18;
	iNumberMeasurementGroups	:	 INT:= 11;
(* System array length *)
	iNumberSystemVar			:	INT := 300;

(* MySQL *)
	gcMySql_iSqlLength			:	 INT := 370; 		(* Defines the size in byte of an array element of "asSqlStatement", used by function blocks "MySql_ExecSql" and "MySql_Query"
															to provide an SQL statement as "ARRAY [0..UpperBound] OF STRING(Size)".*)
	raw_SQL_STR_LENGTH		:	 INT := 350;

	gc_MaxBufferSize 	       :INT := 5000; (*number of items to hold in memory*)
	gv_iBuffCounter			:INT := 0; (* counter for  buffer*)
	gv_iBuffPointer			:INT := 0; (* pointer  for  buffer*)
	gv_Buffer					:ARRAY[0..gc_MaxBufferSize] OF ARRAY[0.. iNumberSystemVar] OF REAL; (*In memory buffer of failed message attempts*)


	gc_sHost : STRING := '### your mysql server address here';  (*'application.dyndns.info';*)
	gc_uiPort : UINT := 3306;
	gc_sUser : STRING := '### your mysql server username ';
	gc_sPwd : STRING := '### your mysql password';
	gc_sDB : STRING := '### your MYSQL database';   	(* Optional - Name of database instance to connect to *)
	gc_sTable:STRING := '### your MYSql table' ;

END_VAR

VAR_GLOBAL PERSISTENT RETAIN

	CurrentRatioPQ1						:	WORD := 400;			(* Current transformer ratio, eg 5 A / 400 A *)
	CurrentRatioPQ2						:	WORD := 400;

END_VAR

(* Data type *)
TYPE typCSV :
STRUCT
	sDescription	:STRING;
	Parameter		:ARRAY[1..gc_ParameterCount] OF STRING;
END_STRUCT
END_TYPE

(* POU 05. System State Array/variables_to_system_array, ST *)
PROGRAM variables_to_system_array
VAR
	i: INT;
	j: INT;
	start : INT;
END_VAR
(* https://docs.google.com/spreadsheets/d/1TR7oXGZyEmNnGigmreKdtnpXsz8mxFcoB4b4beNITCA/edit *)

(* loop trough all variable and measurements groups *)
FOR j := 0 TO iNumberMeasurementGroups-1 DO

	start := j*iNumberMeasurementVar;
	FOR i := 1 TO iNumberMeasurementVar-1  DO

		IF i +start <= iNumberMeasurementVar THEN
			arSystemState[i+start] := arMeasurementsGroup1[i];
		END_IF

		IF i +start > iNumberMeasurementVar AND  i +start <= 2*iNumberMeasurementVar THEN
			arSystemState[i+start] := arMeasurementsGroup2[i];
		END_IF

		IF i +start > 2*iNumberMeasurementVar AND  i +start <= 3*iNumberMeasurementVar THEN
			arSystemState[i+start] := arMeasurementsGroup3[i];
		END_IF

		IF i +start > 3*iNumberMeasurementVar AND  i +start <= 4*iNumberMeasurementVar THEN
			arSystemState[i+start] := arMeasurementsGroup4[i];
		END_IF

		IF i +start > 4*iNumberMeasurementVar AND  i +start <= 5*iNumberMeasurementVar THEN
			arSystemState[i+start] := arMeasurementsGroup5[i];
		END_IF

		IF i +start > 5*iNumberMeasurementVar AND  i +start <= 6*iNumberMeasurementVar THEN
			arSystemState[i+start] := arMeasurementsGroup6[i];
		END_IF

		IF i +start > 6*iNumberMeasurementVar AND  i +start <= 7*iNumberMeasurementVar THEN
			arSystemState[i+start] := arMeasurementsGroup7[i];
		END_IF
		IF i +start > 7*iNumberMeasurementVar AND  i +start <= 8*iNumberMeasurementVar THEN
			arSystemState[i+start] := arMeasurementsGroup8[i];
		END_IF

		IF i +start > 8*iNumberMeasurementVar AND  i +start <= 9*iNumberMeasurementVar THEN
			arSystemState[i+start] := arMeasurementsGroup9[i];
		END_IF

		IF i +start > 9*iNumberMeasurementVar AND  i +start <= 10*iNumberMeasurementVar THEN
			arSystemState[i+start] := arMeasurementsGroupA[i];
		END_IF

		IF i +start > 10*iNumberMeasurementVar AND  i +start <= 11*iNumberMeasurementVar THEN
			arSystemState[i+start] := arMeasurementsGroupB[i];
		END_IF

	END_FOR
END_FOR

(* _____ ALWAYS UDPATE (REVERSRE) THE WRITABLE MODBUS PARAMETERS _____

Bus_Connector_3F_Sync_close_requested_modbus 					: BOOL;
Bus_Connector_3F_Sync_denied_modbus				 				: BOOL;
example:
	Bus_Connector_3F_Sync_close_requested_modbus:=REAL_TO_BOOL(arSystemState[219]);
	Bus_Connector_3F_Sync_denied_modbus :=REAL_TO_BOOL(arSystemState[220]);
*)

(* other system variable*)
arSystemState[199] :=Bus_Connector_L1_P;
arSystemState[200] :=Bus_Connector_L2_P;
arSystemState[201] :=Bus_Connector_L3_P;
arSystemState[202] :=Bus_Connector_L1_Q;
arSystemState[203] :=Bus_Connector_L2_Q;
arSystemState[204] :=Bus_Connector_L3_Q;
arSystemState[205] :=Bus_Connector_L1_V;
arSystemState[206] :=Bus_Connector_L2_V;
arSystemState[207] :=Bus_Connector_L3_V;
arSystemState[208] :=Bus_Connector_L1_I;
arSystemState[209] :=Bus_Connector_L2_I;
arSystemState[210] :=Bus_Connector_L3_I;
arSystemState[211] :=Bus_Connector_L1_f;
arSystemState[212] :=Bus_Connector_L2_f;
arSystemState[213] :=Bus_Connector_L3_f;
arSystemState[214] :=Bus_Connector_3F_radians;
arSystemState[215] :=BOOL_TO_REAL(Bus_Connector_3F_Sync_close_requested);
arSystemState[216] :=BOOL_TO_REAL(Bus_Connector_3F_Sync_closed);
arSystemState[217] :=BOOL_TO_REAL(Bus_Connector_3F_Sync_close_requested_panel);
arSystemState[218] :=BOOL_TO_REAL(Bus_Connector_3F_Sync_denied_panel);
Bus_Connector_3F_Sync_close_requested_modbus:=REAL_TO_BOOL(arSystemState[219]);
Bus_Connector_3F_Sync_denied_modbus :=REAL_TO_BOOL(arSystemState[220]);
arSystemState[221] :=Bus_Connector_3F_Field_Rotation;
arSystemState[222] :=BOOL_TO_REAL(CHP_control_grid_bus_select_controlswitch);
arSystemState[223] :=BOOL_TO_REAL(CHP_control_baterry_bus_select_controlswitch);
arSystemState[224] :=BOOL_TO_REAL(CHP_control_auto_bus_select_controlswitch);
arSystemState[225] :=BOOL_TO_REAL(CHP_control_Offgrid_request);
arSystemState[226] :=CHP_control_Offgrid_Active_Power_control;
arSystemState[227] :=BOOL_TO_REAL(CHP_control_internal_contacter_switch_state);
arSystemState[228] :=EV_control_control_signal;
arSystemState[229] :=Mixer_control_control_signal;
arSystemState[230] :=BOOL_TO_REAL(Group1_3F_Auto_relay_control_battery_bus);
arSystemState[231] :=BOOL_TO_REAL(Group1_3F_Auto_relay_control_grid_bus);
arSystemState[232] :=BOOL_TO_REAL(Group1_3F_Selector_auto_bus_select);
arSystemState[233] :=BOOL_TO_REAL(Group1_3F_relay_state_battery_bus);
arSystemState[234] :=BOOL_TO_REAL(Group1_3F_relay_state_grid_bus);
arSystemState[233] :=BOOL_TO_REAL(Group2_3F_Auto_relay_control_battery_bus);
arSystemState[234] :=BOOL_TO_REAL(Group2_3F_Auto_relay_control_grid_bus);
arSystemState[235] :=BOOL_TO_REAL(Group2_3F_Selector_auto_bus_select);
arSystemState[236] :=BOOL_TO_REAL(Group2_3F_relay_state_battery_bus);
arSystemState[237] :=BOOL_TO_REAL(Group2_3F_relay_state_grid_bus);
arSystemState[236] :=BOOL_TO_REAL(Group3_3F_Auto_relay_control_battery_bus);
arSystemState[237] :=BOOL_TO_REAL(Group3_3F_Auto_relay_control_grid_bus);
arSystemState[238] :=BOOL_TO_REAL(Group3_3F_Selector_auto_bus_select);
arSystemState[239] :=BOOL_TO_REAL(Group3_3F_relay_state_battery_bus);
arSystemState[240] :=BOOL_TO_REAL(Group3_3F_relay_state_grid_bus);
arSystemState[239] :=BOOL_TO_REAL(Group4_3F_Auto_relay_control_battery_bus);
arSystemState[240] :=BOOL_TO_REAL(Group4_3F_Auto_relay_control_grid_bus);
arSystemState[241] :=BOOL_TO_REAL(Group4_3F_Selector_auto_bus_select);
arSystemState[242] :=BOOL_TO_REAL(Group4_3F_relay_state_battery_bus);
arSystemState[243] :=BOOL_TO_REAL(Group4_3F_relay_state_grid_bus);
arSystemState[242] :=BOOL_TO_REAL(Group5_3F_Auto_relay_control_battery_bus);
arSystemState[243] :=BOOL_TO_REAL(Group5_3F_Auto_relay_control_grid_bus);
arSystemState[244] :=BOOL_TO_REAL(Group5_3F_Selector_auto_bus_select);
arSystemState[245] :=BOOL_TO_REAL(Group5_3F_relay_state_battery_bus);
arSystemState[246] :=BOOL_TO_REAL(Group5_3F_relay_state_grid_bus);
arSystemState[245] :=BOOL_TO_REAL(Group6_3F_Auto_relay_control_battery_bus);
arSystemState[246] :=BOOL_TO_REAL(Group6_3F_Auto_relay_control_grid_bus);
arSystemState[247] :=BOOL_TO_REAL(Group6_3F_Selector_auto_bus_select);
arSystemState[248] :=BOOL_TO_REAL(Group6_3F_relay_state_battery_bus);
arSystemState[249] :=BOOL_TO_REAL(Group6_3F_relay_state_grid_bus);
arSystemState[248] :=BOOL_TO_REAL(Group7_3F_Auto_relay_control_battery_bus);
arSystemState[249] :=BOOL_TO_REAL(Group7_3F_Auto_relay_control_grid_bus);
arSystemState[250] :=BOOL_TO_REAL(Group7_3F_Selector_auto_bus_select);
arSystemState[251] :=BOOL_TO_REAL(Group7_3F_relay_state_battery_bus);
arSystemState[252] :=BOOL_TO_REAL(Group7_3F_relay_state_grid_bus);
arSystemState[251] :=BOOL_TO_REAL(Group8_3F_Auto_relay_control_battery_bus);
arSystemState[252] :=BOOL_TO_REAL(Group8_3F_Auto_relay_control_grid_bus);
arSystemState[253] :=BOOL_TO_REAL(Group8_3F_Selector_auto_bus_select);
arSystemState[254] :=BOOL_TO_REAL(Group8_3F_relay_state_battery_bus);
arSystemState[255] :=BOOL_TO_REAL(Group8_3F_relay_state_grid_bus);
arSystemState[256] :=BOOL_TO_REAL(Group9_3F_Auto_relay_control_battery_bus);
arSystemState[257] :=BOOL_TO_REAL(Group9_3F_Auto_relay_control_grid_bus);
arSystemState[258] :=BOOL_TO_REAL(Group9_3F_Selector_auto_bus_select);
arSystemState[259] :=BOOL_TO_REAL(Group9_3F_relay_state_battery_bus);
arSystemState[260] :=BOOL_TO_REAL(Group9_3F_relay_state_grid_bus);
arSystemState[261] :=Group_control_Frequencybased_bus_selecting_state;
arSystemState[262] :=Group_control_min_time_above_switch_frequency;
arSystemState[263] :=Group_control_min_time_below_switch_frequency;
arSystemState[264] :=Group1_3F_Switch_frequency_to_batterybus;
arSystemState[265] :=Group1_3F_Switch_frequency_to_gridbus;
arSystemState[266] :=Group1_3F_min_time_between_switching;
arSystemState[267] :=Group2_3F_Switch_frequency_to_batterybus;
arSystemState[268] :=Group2_3F_Switch_frequency_to_gridbus;
arSystemState[269] :=Group2_3F_min_time_between_switching;
arSystemState[268] :=Group3_3F_Switch_frequency_to_batterybus;
arSystemState[269] :=Group3_3F_Switch_frequency_to_gridbus;
arSystemState[270] :=Group3_3F_min_time_between_switching;
arSystemState[271] :=Group4_3F_Switch_frequency_to_batterybus;
arSystemState[270] :=Group4_3F_Switch_frequency_to_gridbus;
arSystemState[271] :=Group4_3F_min_time_between_switching;
arSystemState[272] :=Group5_3F_Switch_frequency_to_batterybus;
arSystemState[273] :=Group5_3F_Switch_frequency_to_gridbus;
arSystemState[272] :=Group5_3F_min_time_between_switching;
arSystemState[273] :=Group6_3F_Switch_frequency_to_batterybus;
arSystemState[274] :=Group6_3F_Switch_frequency_to_gridbus;
arSystemState[275] :=Group6_3F_min_time_between_switching;
arSystemState[274] :=Group7_3F_Switch_frequency_to_batterybus;
arSystemState[275] :=Group7_3F_Switch_frequency_to_gridbus;
arSystemState[276] :=Group7_3F_min_time_between_switching;
arSystemState[277] :=Group8_3F_Switch_frequency_to_batterybus;
arSystemState[276] :=Group8_3F_Switch_frequency_to_gridbus;
arSystemState[277] :=Group8_3F_min_time_between_switching;
arSystemState[278] :=Group9_3F_Switch_frequency_to_batterybus;
arSystemState[279] :=Group9_3F_Switch_frequency_to_gridbus;
arSystemState[278] :=Group9_3F_min_time_between_switching;
arSystemState[279] :=BOOL_TO_REAL(Control_panel_status_warning_led);
arSystemState[280] :=BOOL_TO_REAL(Control_panel_status_error_led);
arSystemState[281] :=BOOL_TO_REAL(Control_panel_status_operational_led);
END_PROGRAM

(* POU 03. Synchroniser Switch control/SynchroniserSwitch, LD *)
PROGRAM SynchroniserSwitch
VAR
END_VAR
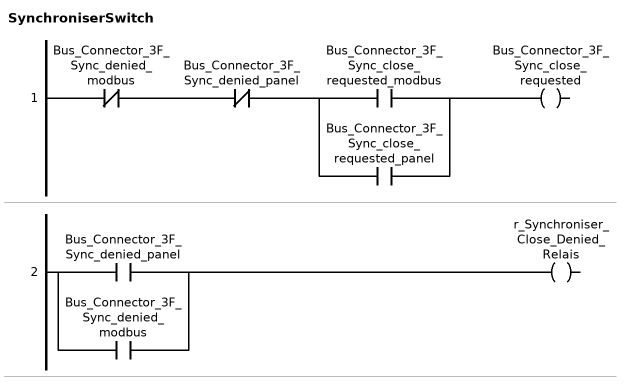
_LD_ (* Ladder Diagram *)
NETWORK 1
	[/Bus_Connector_3F_Sync_denied_modbus] - [/Bus_Connector_3F_Sync_denied_panel] - { [Bus_Connector_3F_Sync_close_requested_modbus] | [Bus_Connector_3F_Sync_close_requested_panel] } --- (Bus_Connector_3F_Sync_close_requested)
NETWORK 2
	{ [Bus_Connector_3F_Sync_denied_panel] | [Bus_Connector_3F_Sync_denied_modbus] } --- (r_Synchroniser_Close_Denied_Relais)
_END_LD_
(* the same logic as Structured Text *)
(* Network 1 *)
Bus_Connector_3F_Sync_close_requested := NOT Bus_Connector_3F_Sync_denied_modbus AND NOT Bus_Connector_3F_Sync_denied_panel AND (Bus_Connector_3F_Sync_close_requested_modbus OR Bus_Connector_3F_Sync_close_requested_panel);
(* Network 2 *)
r_Synchroniser_Close_Denied_Relais := Bus_Connector_3F_Sync_denied_panel OR Bus_Connector_3F_Sync_denied_modbus;
END_PROGRAM

(* POU 04. Frequency based Bus Select/Group2, FBD *)
PROGRAM Group2
VAR
	Switch2:fbSwitchRelaysBatOrGridBus;
END_VAR
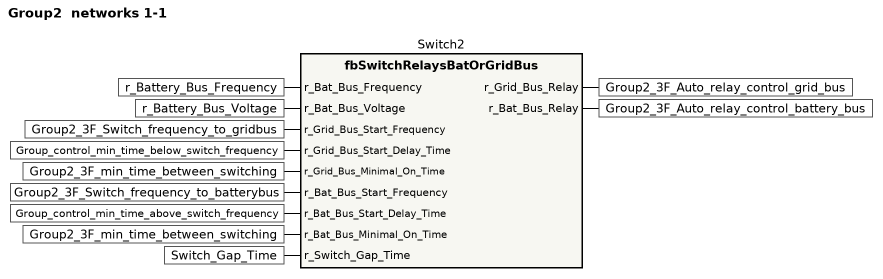
_FBD_ (* Function Block Diagram *)
NETWORK 1
	Switch2:fbSwitchRelaysBatOrGridBus(r_Bat_Bus_Frequency: r_Battery_Bus_Frequency, r_Bat_Bus_Voltage: r_Battery_Bus_Voltage, r_Grid_Bus_Start_Frequency: Group2_3F_Switch_frequency_to_gridbus, r_Grid_Bus_Start_Delay_Time: Group_control_min_time_below_switch_frequency, r_Grid_Bus_Minimal_On_Time: Group2_3F_min_time_between_switching, r_Bat_Bus_Start_Frequency: Group2_3F_Switch_frequency_to_batterybus, r_Bat_Bus_Start_Delay_Time: Group_control_min_time_above_switch_frequency, r_Bat_Bus_Minimal_On_Time: Group2_3F_min_time_between_switching, r_Switch_Gap_Time: Switch_Gap_Time, r_Bat_Bus_Relay => Group2_3F_Auto_relay_control_battery_bus) => Group2_3F_Auto_relay_control_grid_bus
_END_FBD_
(* the same logic as Structured Text *)
(* Network 1 *)
Switch2(r_Bat_Bus_Frequency := r_Battery_Bus_Frequency, r_Bat_Bus_Voltage := r_Battery_Bus_Voltage, r_Grid_Bus_Start_Frequency := Group2_3F_Switch_frequency_to_gridbus, r_Grid_Bus_Start_Delay_Time := Group_control_min_time_below_switch_frequency, r_Grid_Bus_Minimal_On_Time := Group2_3F_min_time_between_switching, r_Bat_Bus_Start_Frequency := Group2_3F_Switch_frequency_to_batterybus, r_Bat_Bus_Start_Delay_Time := Group_control_min_time_above_switch_frequency, r_Bat_Bus_Minimal_On_Time := Group2_3F_min_time_between_switching, r_Switch_Gap_Time := Switch_Gap_Time);
Group2_3F_Auto_relay_control_battery_bus := Switch2.r_Bat_Bus_Relay;
Group2_3F_Auto_relay_control_grid_bus := Switch2.r_Grid_Bus_Relay;
END_PROGRAM

(* POU 04. Frequency based Bus Select/fbSwitchRelaysBatOrGridBus, SFC *)
FUNCTION_BLOCK fbSwitchRelaysBatOrGridBus
VAR_INPUT

	r_Bat_Bus_Frequency						:	REAL;
	r_Bat_Bus_Voltage							:	REAL;
	r_Grid_Bus_Start_Frequency						:	REAL;
	r_Grid_Bus_Start_Delay_Time					:	REAL;
	r_Grid_Bus_Minimal_On_Time					:	REAL;
	r_Bat_Bus_Start_Frequency					:	REAL;
	r_Bat_Bus_Start_Delay_Time				:	REAL;
	r_Bat_Bus_Minimal_On_Time				:	REAL;
	r_Switch_Gap_Time								: 	REAL;		(* Time between on and off grid relay switching (dead bus gap) *)

END_VAR
VAR_OUTPUT

	r_Grid_Bus_Relay								:	BOOL;
	r_Bat_Bus_Relay									:	BOOL;

END_VAR
VAR
	r_Bat_Bus_Min_Voltage 							: 	REAL :=200;
	r_Checked_Grid_Bus_Start_Frequency			:	REAL;
	r_Checked_Bat_Bus_Start_Frequency			:	REAL;

	t_Grid_Bus_Start_Delay_Timer					:	TON;
	t_Bat_Bus_Start_Delay_Timer					:	TON;


(*	t_Bat_Bus_Start_Delay_Timer: BOOL;*)
END_VAR
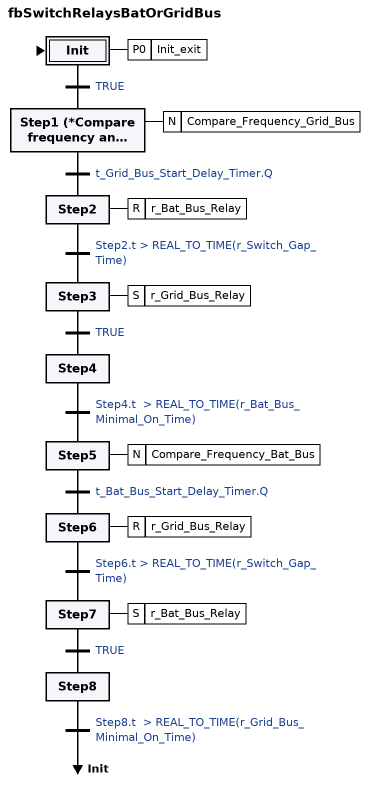
INITIAL_STEP Init:
	Init_exit(P0);
END_STEP
TRANSITION FROM Init TO Step1 (*Compare frequency and voltage *) := TRUE;
END_TRANSITION
STEP Step1 (*Compare frequency and voltage *):
	Compare_Frequency_Grid_Bus(N);
END_STEP
TRANSITION FROM Step1 (*Compare frequency and voltage *) TO Step2 := t_Grid_Bus_Start_Delay_Timer.Q;
END_TRANSITION
STEP Step2:
	r_Bat_Bus_Relay(R);
END_STEP
TRANSITION FROM Step2 TO Step3 := Step2.t > REAL_TO_TIME(r_Switch_Gap_Time);
END_TRANSITION
STEP Step3:
	r_Grid_Bus_Relay(S);
END_STEP
TRANSITION FROM Step3 TO Step4 := TRUE;
END_TRANSITION
STEP Step4:
END_STEP
TRANSITION FROM Step4 TO Step5 := Step4.t  > REAL_TO_TIME(r_Bat_Bus_Minimal_On_Time);
END_TRANSITION
STEP Step5:
	Compare_Frequency_Bat_Bus(N);
END_STEP
TRANSITION FROM Step5 TO Step6 := t_Bat_Bus_Start_Delay_Timer.Q;
END_TRANSITION
STEP Step6:
	r_Grid_Bus_Relay(R);
END_STEP
TRANSITION FROM Step6 TO Step7 := Step6.t > REAL_TO_TIME(r_Switch_Gap_Time);
END_TRANSITION
STEP Step7:
	r_Bat_Bus_Relay(S);
END_STEP
TRANSITION FROM Step7 TO Step8 := TRUE;
END_TRANSITION
STEP Step8:
END_STEP
TRANSITION FROM Step8 TO Init := Step8.t  > REAL_TO_TIME(r_Grid_Bus_Minimal_On_Time);
END_TRANSITION

ACTION Init_exit:
(* Off grid frequency should by higher than on grid frequency to prevent pendel behaviour of states *)

IF r_Bat_Bus_Start_Frequency > r_Grid_Bus_Start_Frequency THEN

	r_Checked_Bat_Bus_Start_Frequency := r_Bat_Bus_Start_Frequency;
	r_Checked_Grid_Bus_Start_Frequency := r_Grid_Bus_Start_Frequency;

ELSE

	r_Checked_Bat_Bus_Start_Frequency := r_Bat_Bus_Start_Frequency;
	r_Checked_Grid_Bus_Start_Frequency := r_Bat_Bus_Start_Frequency;

END_IF
END_ACTION
END_FUNCTION_BLOCK
ACTION Compare_Frequencies:
(* Bat_Bus start frequency should by higher than grid bus start frequency to prevent pendel behaviour of states *)

IF r_Bat_Bus_Start_Frequency > r_Grid_Bus_Start_Frequency THEN

	r_Checked_Bat_Bus_Start_Frequency := r_Bat_Bus_Start_Frequency;
	r_Checked_Grid_Bus_Start_Frequency := r_Grid_Bus_Start_Frequency;

ELSE

	r_Checked_Bat_Bus_Start_Frequency := r_Bat_Bus_Start_Frequency;
	r_Checked_Grid_Bus_Start_Frequency := r_Bat_Bus_Start_Frequency;

END_IF
END_ACTION
ACTION Compare_Frequency_Bat_Bus:
t_Bat_Bus_Start_Delay_Timer(
	IN:= r_Bat_Bus_Frequency > r_Checked_Bat_Bus_Start_Frequency AND r_Bat_Bus_Voltage > r_Bat_Bus_Min_Voltage,
	PT:= REAL_TO_TIME(r_Grid_Bus_Start_Delay_Time));
END_ACTION
ACTION Compare_Frequency_Grid_Bus:
t_Grid_Bus_Start_Delay_Timer(
	IN:= r_Bat_Bus_Frequency < r_Checked_Grid_Bus_Start_Frequency,
	PT:= REAL_TO_TIME(r_Grid_Bus_Start_Delay_Time));
END_ACTION

(* POU 04. Frequency based Bus Select/init, ST *)
PROGRAM init
VAR
END_VAR
(* frequency based switching is deactivated BY default AND can be activated via modbus *)

arSystemState[246] :=Group_control_Frequencybased_bus_selecting_state;  (* default is off *)
arSystemState[247] :=Group_control_min_time_above_switch_frequency;
arSystemState[248] :=Group_control_min_time_below_switch_frequency;
arSystemState[249] :=Group1_3F_Switch_frequency_to_batterybus;
arSystemState[250] :=Group1_3F_Switch_frequency_to_gridbus;
arSystemState[251] :=Group1_3F_min_time_between_switching;
arSystemState[252] :=Group2_3F_Switch_frequency_to_batterybus;
arSystemState[253] :=Group2_3F_Switch_frequency_to_gridbus;
arSystemState[254] :=Group2_3F_min_time_between_switching;
arSystemState[253] :=Group3_3F_Switch_frequency_to_batterybus;
arSystemState[254] :=Group3_3F_Switch_frequency_to_gridbus;
arSystemState[255] :=Group3_3F_min_time_between_switching;
arSystemState[256] :=Group4_3F_Switch_frequency_to_batterybus;
arSystemState[255] :=Group4_3F_Switch_frequency_to_gridbus;
arSystemState[256] :=Group4_3F_min_time_between_switching;
arSystemState[257] :=Group5_3F_Switch_frequency_to_batterybus;
arSystemState[258] :=Group5_3F_Switch_frequency_to_gridbus;
arSystemState[257] :=Group5_3F_min_time_between_switching;
arSystemState[258] :=Group6_3F_Switch_frequency_to_batterybus;
arSystemState[259] :=Group6_3F_Switch_frequency_to_gridbus;
arSystemState[260] :=Group6_3F_min_time_between_switching;
arSystemState[259] :=Group7_3F_Switch_frequency_to_batterybus;
arSystemState[260] :=Group7_3F_Switch_frequency_to_gridbus;
arSystemState[261] :=Group7_3F_min_time_between_switching;
arSystemState[262] :=Group8_3F_Switch_frequency_to_batterybus;
arSystemState[261] :=Group8_3F_Switch_frequency_to_gridbus;
arSystemState[262] :=Group8_3F_min_time_between_switching;
arSystemState[263] :=Group9_3F_Switch_frequency_to_batterybus;
arSystemState[264] :=Group9_3F_Switch_frequency_to_gridbus;
arSystemState[263] :=Group9_3F_min_time_between_switching;
END_PROGRAM

(* POU 08. SD CARD logging/WRITE_CSV/WRITE_DATA, FBD *)
PROGRAM WRITE_DATA
VAR
	FB1				: FbDatalogger;
	xGo				: BOOL		:= TRUE;
	xTrigger			: BOOL;
	Channels			: ARRAY [1.. 80] OF typUserInput;
	Settings			: typConfigDatalogger;
	bDType			: BYTE := 1;
	xFirstCycle			: BOOL := TRUE;
	i: INT;

END_VAR
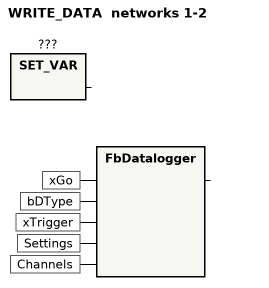
_FBD_ (* Function Block Diagram *)
NETWORK 1
	???:SET_VAR()
NETWORK 2
	FbDatalogger(xGo, bDType, xTrigger, Settings, Channels)
_END_FBD_
(* the same logic as Structured Text *)
(* Network 1: see the listing above *)
(* Network 2 *)
FbDatalogger(xGo, bDType, xTrigger, Settings, Channels);
END_PROGRAM
ACTION SET_VAR:
IF xFirstCycle THEN

	settings.bInterval					:= 3; 						(* 1 = hour, 2= minutes, 3 = seconds *)
	settings.iIntervalFactor			:= 5;						(* number of hours/minutes/seconds, depending on choice b.Interval *)
	settings.sFilename				:= 'Meetdata.csv';				(* Filename csv-file *)
	settings.sPath						:= '/media/sd/';				(* Path where the csv-file is stored *)
	settings.xAppendDate			:= TRUE;					(* When true, the date on the controller is added to the filename*)
	settings.xCyclicLogging			:= TRUE;					(* When true, information is stored cyclic on the controller/SD card *)

	Channels[1].xChannelExists		:= TRUE;
	Channels[1].sChannelName		:= 'PhaseCurrentl2';
	Channels[1].sUnit					:= 'A';
	Channels[1].rAlarmLowerLimit	:= -10000000;
	Channels[1].rAlarmUpperLimit	:= 10000000;

	Channels[2].xChannelExists		:= TRUE;
	Channels[2].sChannelName		:= 'VoltageV31';
	Channels[2].sUnit					:= 'V';
	Channels[2].rAlarmLowerLimit	:= -10000000;
	Channels[2].rAlarmUpperLimit	:= 10000000;

	Channels[3].xChannelExists		:= TRUE;
	Channels[3].sChannelName		:= 'Pactive';
	Channels[3].sUnit					:= 'W';
	Channels[3].rAlarmLowerLimit	:= -10000000;
	Channels[3].rAlarmUpperLimit	:= 10000000;

	Channels[4].xChannelExists		:= TRUE;
	Channels[4].sChannelName		:= 'Preactive';
	Channels[4].sUnit					:= 'VAr';;
	Channels[4].rAlarmLowerLimit	:= -10000000;
	Channels[4].rAlarmUpperLimit	:= 10000000;

	Channels[5].xChannelExists		:= TRUE;
	Channels[5].sChannelName		:= 'ShortCircuitDirectionA';
	Channels[5].sUnit					:= ' ';
	Channels[5].rAlarmLowerLimit	:= -10000000;
	Channels[5].rAlarmUpperLimit	:= 10000000;

	Channels[6].xChannelExists		:= TRUE;
	Channels[6].sChannelName		:= 'ShortCircuitDirectionB';
	Channels[6].sUnit					:= ' ';
	Channels[6].rAlarmLowerLimit	:= -10000000;
	Channels[6].rAlarmUpperLimit	:= 10000000;

	Channels[7].xChannelExists		:= TRUE;
	Channels[7].sChannelName		:= 'Phase1';
	Channels[7].sUnit					:= ' ';
	Channels[7].rAlarmLowerLimit	:= -10000000;
	Channels[7].rAlarmUpperLimit	:= 10000000;

	Channels[8].xChannelExists		:= TRUE;
	Channels[8].sChannelName		:= 'Phase2';
	Channels[8].sUnit					:=  ' ';
	Channels[8].rAlarmLowerLimit	:= -10000000;
	Channels[8].rAlarmUpperLimit	:= 10000000;

	Channels[9].xChannelExists		:= TRUE;
	Channels[9].sChannelName		:= 'Phase3';
	Channels[9].sUnit					:=  ' ';
	Channels[9].rAlarmLowerLimit	:= -10000000;
	Channels[9].rAlarmUpperLimit	:= 10000000;

	Channels[10].xChannelExists		:= TRUE;
	Channels[10].sChannelName		:= 'StatusRemoteSwitching';
	Channels[10].sUnit					:=  ' ';
	Channels[10].rAlarmLowerLimit	:= -10000000;
	Channels[10].rAlarmUpperLimit	:= 10000000;


	Channels[11].xChannelExists		:= TRUE;
	Channels[11].sChannelName		:= 'SwitchLoadBreaker';
	Channels[11].sUnit					:=  ' ';
	Channels[11].rAlarmLowerLimit	:= -10000000;
	Channels[11].rAlarmUpperLimit	:= 10000000;

	Channels[12].xChannelExists		:= TRUE;
	Channels[12].sChannelName		:= 'Bay3CurrentL1';
	Channels[12].sUnit					:=  'A ';
	Channels[12].rAlarmLowerLimit	:= -10000000;
	Channels[12].rAlarmUpperLimit	:= 10000000;

	Channels[13].xChannelExists		:= TRUE;
	Channels[13].sChannelName		:= 'Bay3CurrentL2';
	Channels[13].sUnit					:=  'A ';
	Channels[13].rAlarmLowerLimit	:= -10000000;
	Channels[13].rAlarmUpperLimit	:= 10000000;

	Channels[14].xChannelExists		:= TRUE;
	Channels[14].sChannelName		:= 'Bay3CurrentL3';
	Channels[14].sUnit					:=  'A ';
	Channels[14].rAlarmLowerLimit	:= -10000000;
	Channels[14].rAlarmUpperLimit	:= 10000000;

	Channels[15].xChannelExists		:= TRUE;
	Channels[15].sChannelName		:= 'Bay4CurrentL1';
	Channels[15].sUnit					:=  'A ';
	Channels[15].rAlarmLowerLimit	:= -10000000;
	Channels[15].rAlarmUpperLimit	:= 10000000;

	Channels[16].xChannelExists		:= TRUE;
	Channels[16].sChannelName		:= 'Bay4CurrentL2';
	Channels[16].sUnit					:=  'A ';
	Channels[16].rAlarmLowerLimit	:= -10000000;
	Channels[16].rAlarmUpperLimit	:= 10000000;

	Channels[17].xChannelExists		:= TRUE;
	Channels[17].sChannelName		:= 'Bay4CurrentL3';
	Channels[17].sUnit					:=  'A ';
	Channels[17].rAlarmLowerLimit	:= -10000000;
	Channels[17].rAlarmUpperLimit	:= 10000000;

	xFirstCycle := FALSE;

END_IF

	Channels[1].rValue			:= MBCFG_ModbusSlave.PhaseCurrenL2;
	Channels[2].rValue			:= MBCFG_ModbusSlave.VoltageV31;
	Channels[3].rValue			:= MBCFG_ModbusSlave.Pactive;
	Channels[4].rValue			:= MBCFG_ModbusSlave.Preactive;
	Channels[5].rValue			:= MBCFG_ModbusSlave.ShortCircuitA;
	Channels[6].rValue			:= MBCFG_ModbusSlave.ShortCircuitB;
	Channels[7].rValue			:= MBCFG_ModbusSlave.Phase1;
	Channels[8].rValue			:= MBCFG_ModbusSlave.Phase2;
	Channels[9].rValue			:= MBCFG_ModbusSlave.Phase3;
	Channels[10].rValue			:= MBCFG_ModbusSlave.StatusRemoteSwitching;
	Channels[11].rValue			:= MBCFG_ModbusSlave.SwitchLoadBreaker;
	Channels[12].rValue			:= PQ_1.arCurrent[1];
	Channels[13].rValue			:= PQ_1.arCurrent[2];
	Channels[14].rValue			:= PQ_1.arCurrent[3];
	Channels[15].rValue			:= PQ_2.arCurrent[1];
	Channels[16].rValue			:= PQ_2.arCurrent[2];
	Channels[17].rValue			:= PQ_2.arCurrent[3];





(* For-loop to set the channels to be written on the SD-card *)
END_ACTION

(* POU 01. PowerQualityMeasurements/PQ_1, FBD *)
PROGRAM PQ_1
VAR
	abProcessImageInput	AT %IW12			: ARRAY[0..23] OF BYTE;
	abProcessImageOutput 	AT %QW20		: ARRAY[0..23] OF BYTE;

	bToken										: BYTE;

	State_750_495 							: Fb_750_495_State;
		typ_750_495_State 						: typ_750_495_State;

	Configuration_750_495					: Fb_750_495_Configuration;
		typConfig_750_495						: typConfig_750_495;
		xReadyConfig								: BOOL;
		bFeedbackConfig							: BYTE;

	AC_Compact_01_750_495				: Fb_750_495_AC_Compact_01;
		rTotalActivePower							: REAL;
		rTotalReactivePower						: REAL;
		rTotalApparentPower						: REAL;
		rTotalPowerFactorPF						: REAL;
		rTotalActiveEnergy							: REAL;
		rTotalReactiveEnergy						: REAL;
		rTotalApparentEnergy						: REAL;
		rCurrentN									: REAL;
		xRotatingField								: BOOL;
		arCurrent									: ARRAY[1..3] OF REAL;
		axOvercurrent								: ARRAY[1..3] OF BOOL;
		arVoltage_L_N							: ARRAY[1..3] OF REAL;
		axUndervoltage							: ARRAY[1..3] OF BOOL;
		axOvervoltage								: ARRAY[1..3] OF BOOL;
		arActivePower								: ARRAY[1..3] OF REAL;
		arReactivePower							: ARRAY[1..3] OF REAL;
		arApparentPower							: ARRAY[1..3] OF REAL;
		arCosPhi									: ARRAY[1..3] OF REAL;
		arPowerFactorPF							: ARRAY[1..3] OF REAL;
		arFrequency								: ARRAY[1..3] OF REAL;
		axNoZero									: ARRAY[1..3] OF BOOL;
		axVoltSag									: ARRAY[1..3] OF BOOL;
		ai4Quadrant								: ARRAY[1..3] OF INT;

		xReadyCompact_01						: BOOL;
		abFeedbackCompact_01					: ARRAY[1..8] OF BYTE;


END_VAR
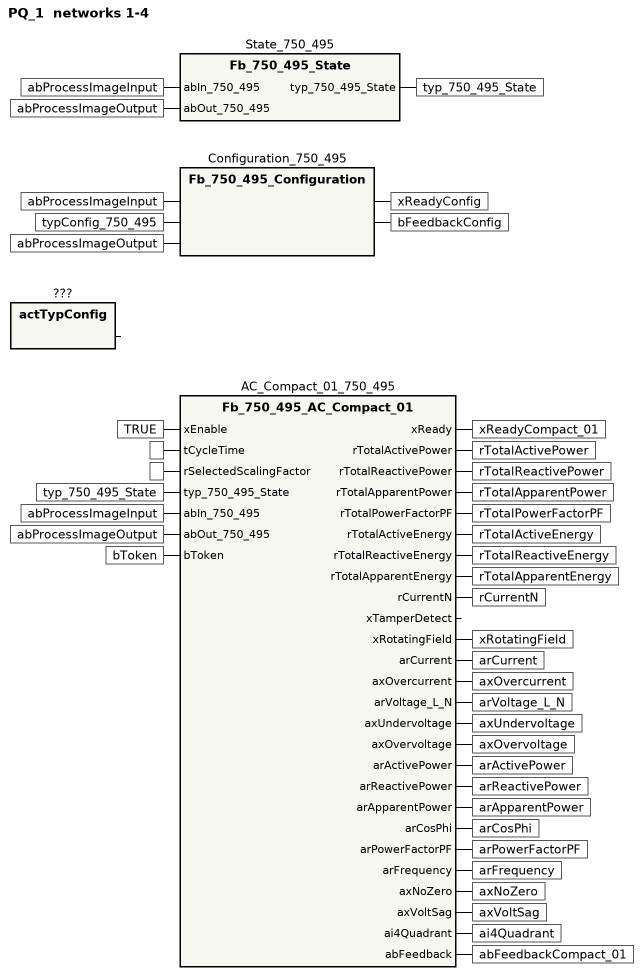
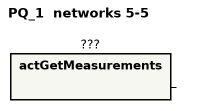
_FBD_ (* Function Block Diagram *)
NETWORK 1
	State_750_495:Fb_750_495_State(abIn_750_495: abProcessImageInput, abOut_750_495: abProcessImageOutput) => typ_750_495_State
NETWORK 2
	Configuration_750_495:Fb_750_495_Configuration(abProcessImageInput, typConfig_750_495, abProcessImageOutput, out 2 => bFeedbackConfig) => xReadyConfig
NETWORK 3
	???:actTypConfig()
NETWORK 4
	AC_Compact_01_750_495:Fb_750_495_AC_Compact_01(xEnable: TRUE, tCycleTime: , rSelectedScalingFactor: , typ_750_495_State: typ_750_495_State, abIn_750_495: abProcessImageInput, abOut_750_495: abProcessImageOutput, bToken: bToken, rTotalActivePower => rTotalActivePower, rTotalReactivePower => rTotalReactivePower, rTotalApparentPower => rTotalApparentPower, rTotalPowerFactorPF => rTotalPowerFactorPF, rTotalActiveEnergy => rTotalActiveEnergy, rTotalReactiveEnergy => rTotalReactiveEnergy, rTotalApparentEnergy => rTotalApparentEnergy, rCurrentN => rCurrentN, xRotatingField => xRotatingField, arCurrent => arCurrent, axOvercurrent => axOvercurrent, arVoltage_L_N => arVoltage_L_N, axUndervoltage => axUndervoltage, axOvervoltage => axOvervoltage, arActivePower => arActivePower, arReactivePower => arReactivePower, arApparentPower => arApparentPower, arCosPhi => arCosPhi, arPowerFactorPF => arPowerFactorPF, arFrequency => arFrequency, axNoZero => axNoZero, axVoltSag => axVoltSag, ai4Quadrant => ai4Quadrant, abFeedback => abFeedbackCompact_01) => xReadyCompact_01
NETWORK 5
	???:actGetMeasurements()
_END_FBD_
(* the same logic as Structured Text *)
(* Network 1 *)
State_750_495(abIn_750_495 := abProcessImageInput, abOut_750_495 := abProcessImageOutput);
typ_750_495_State := State_750_495.typ_750_495_State;
(* Network 2: see the listing above *)
(* Network 3: see the listing above *)
(* Network 4: see the listing above *)
(* Network 5: see the listing above *)
END_PROGRAM
ACTION actGetMeasurements:
arMeasurementsGroup1[1] := arActivePower[1];
arMeasurementsGroup1[2] := arActivePower[2];
arMeasurementsGroup1[3] := arActivePower[3];
arMeasurementsGroup1[4] := arReactivePower[1];
arMeasurementsGroup1[5] := arReactivePower[2];
arMeasurementsGroup1[6] := arReactivePower[3];
arMeasurementsGroup1[7] := arVoltage_L_N[1];
arMeasurementsGroup1[8] := arVoltage_L_N[2];
arMeasurementsGroup1[9] := arVoltage_L_N[3];
arMeasurementsGroup1[10] := arCurrent[1];
arMeasurementsGroup1[11] := arCurrent[2];
arMeasurementsGroup1[12] := arCurrent[3];
arMeasurementsGroup1[13] := arFrequency[1];
arMeasurementsGroup1[14] := arFrequency[2];
arMeasurementsGroup1[15] := arFrequency[3];
arMeasurementsGroup1[16] := rTotalActiveEnergy;
arMeasurementsGroup1[17] := BOOL_TO_REAL(xRotatingField);
arMeasurementsGroup1[18] := rTotalReactiveEnergy;
END_ACTION
ACTION actTypConfig:
typConfig_750_495.typChannelConfig[1].xEnableUserScaling:= TRUE;
typConfig_750_495.typChannelConfig[1].wCurrentTransformerRatio :=CurrentRatioPQ1;

typConfig_750_495.typChannelConfig[2].xEnableUserScaling:= TRUE;
typConfig_750_495.typChannelConfig[2].wCurrentTransformerRatio :=CurrentRatioPQ1;

typConfig_750_495.typChannelConfig[3].xEnableUserScaling:= TRUE;
typConfig_750_495.typChannelConfig[3].wCurrentTransformerRatio :=CurrentRatioPQ1;

typConfig_750_495.xWriteConfig := TRUE;
END_ACTION

(* POU 01. PowerQualityMeasurements/PQ_2, FBD *)
PROGRAM PQ_2
VAR
	abProcessImageInput	AT %IW24			: ARRAY[0..23] OF BYTE;
	abProcessImageOutput 	AT %QW32 			: ARRAY[0..23] OF BYTE;

	bToken										: BYTE;

	State_750_495 							: Fb_750_495_State;
		typ_750_495_State 						: typ_750_495_State;

	Configuration_750_495					: Fb_750_495_Configuration;
		typConfig_750_495						: typConfig_750_495;
		xReadyConfig								: BOOL;
		bFeedbackConfig							: BYTE;

	AC_Compact_01_750_495				: Fb_750_495_AC_Compact_01;
		rTotalActivePower							: REAL;
		rTotalReactivePower						: REAL;
		rTotalApparentPower						: REAL;
		rTotalPowerFactorPF						: REAL;
		rTotalActiveEnergy							: REAL;
		rTotalReactiveEnergy						: REAL;
		rTotalApparentEnergy						: REAL;
		rCurrentN									: REAL;
		xRotatingField								: BOOL;
		arCurrent									: ARRAY[1..3] OF REAL;
		axOvercurrent								: ARRAY[1..3] OF BOOL;
		arVoltage_L_N							: ARRAY[1..3] OF REAL;
		axUndervoltage							: ARRAY[1..3] OF BOOL;
		axOvervoltage								: ARRAY[1..3] OF BOOL;
		arActivePower								: ARRAY[1..3] OF REAL;
		arReactivePower							: ARRAY[1..3] OF REAL;
		arApparentPower							: ARRAY[1..3] OF REAL;
		arCosPhi									: ARRAY[1..3] OF REAL;
		arPowerFactorPF							: ARRAY[1..3] OF REAL;
		arFrequency								: ARRAY[1..3] OF REAL;
		axNoZero									: ARRAY[1..3] OF BOOL;
		axVoltSag									: ARRAY[1..3] OF BOOL;
		ai4Quadrant								: ARRAY[1..3] OF INT;

		xReadyCompact_01						: BOOL;
		abFeedbackCompact_01					: ARRAY[1..8] OF BYTE;


END_VAR
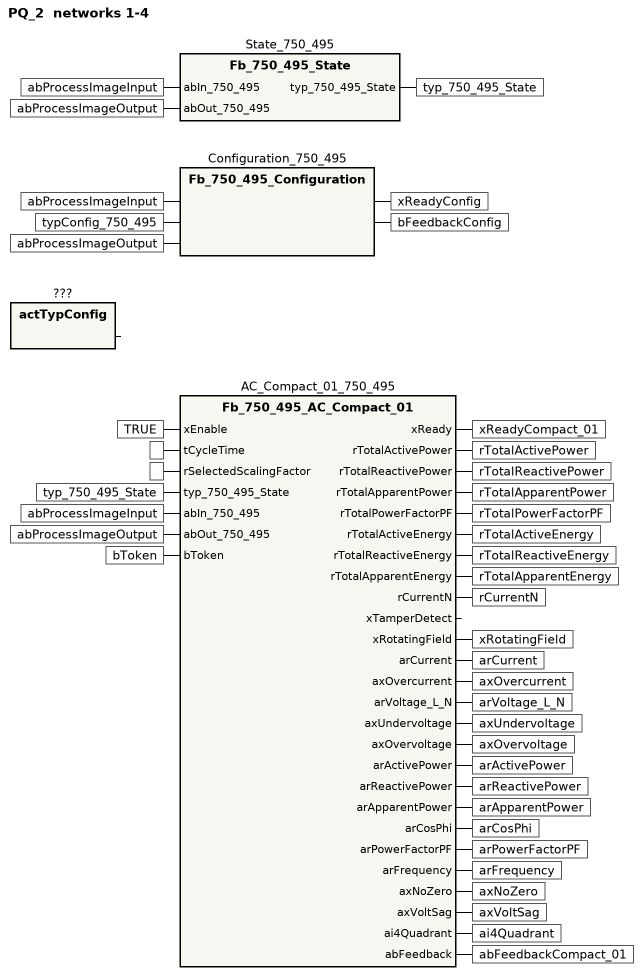
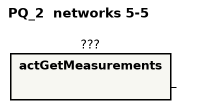
_FBD_ (* Function Block Diagram *)
NETWORK 1
	State_750_495:Fb_750_495_State(abIn_750_495: abProcessImageInput, abOut_750_495: abProcessImageOutput) => typ_750_495_State
NETWORK 2
	Configuration_750_495:Fb_750_495_Configuration(abProcessImageInput, typConfig_750_495, abProcessImageOutput, out 2 => bFeedbackConfig) => xReadyConfig
NETWORK 3
	???:actTypConfig()
NETWORK 4
	AC_Compact_01_750_495:Fb_750_495_AC_Compact_01(xEnable: TRUE, tCycleTime: , rSelectedScalingFactor: , typ_750_495_State: typ_750_495_State, abIn_750_495: abProcessImageInput, abOut_750_495: abProcessImageOutput, bToken: bToken, rTotalActivePower => rTotalActivePower, rTotalReactivePower => rTotalReactivePower, rTotalApparentPower => rTotalApparentPower, rTotalPowerFactorPF => rTotalPowerFactorPF, rTotalActiveEnergy => rTotalActiveEnergy, rTotalReactiveEnergy => rTotalReactiveEnergy, rTotalApparentEnergy => rTotalApparentEnergy, rCurrentN => rCurrentN, xRotatingField => xRotatingField, arCurrent => arCurrent, axOvercurrent => axOvercurrent, arVoltage_L_N => arVoltage_L_N, axUndervoltage => axUndervoltage, axOvervoltage => axOvervoltage, arActivePower => arActivePower, arReactivePower => arReactivePower, arApparentPower => arApparentPower, arCosPhi => arCosPhi, arPowerFactorPF => arPowerFactorPF, arFrequency => arFrequency, axNoZero => axNoZero, axVoltSag => axVoltSag, ai4Quadrant => ai4Quadrant, abFeedback => abFeedbackCompact_01) => xReadyCompact_01
NETWORK 5
	???:actGetMeasurements()
_END_FBD_
(* the same logic as Structured Text *)
(* Network 1 *)
State_750_495(abIn_750_495 := abProcessImageInput, abOut_750_495 := abProcessImageOutput);
typ_750_495_State := State_750_495.typ_750_495_State;
(* Network 2: see the listing above *)
(* Network 3: see the listing above *)
(* Network 4: see the listing above *)
(* Network 5: see the listing above *)
END_PROGRAM
ACTION actGetMeasurements:
arMeasurementsGroup2[1] := arActivePower[1];
arMeasurementsGroup2[2] := arActivePower[2];
arMeasurementsGroup2[3] := arActivePower[3];
arMeasurementsGroup2[4] := arReactivePower[1];
arMeasurementsGroup2[5] := arReactivePower[2];
arMeasurementsGroup2[6] := arReactivePower[3];
arMeasurementsGroup2[7] := arVoltage_L_N[1];
arMeasurementsGroup2[8] := arVoltage_L_N[2];
arMeasurementsGroup2[9] := arVoltage_L_N[3];
arMeasurementsGroup2[10] := arCurrent[1];
arMeasurementsGroup2[11] := arCurrent[2];
arMeasurementsGroup2[12] := arCurrent[3];
arMeasurementsGroup2[13] := arFrequency[1];
arMeasurementsGroup2[14] := arFrequency[2];
arMeasurementsGroup2[15] := arFrequency[3];
arMeasurementsGroup2[16] := rTotalActiveEnergy;
arMeasurementsGroup2[17] := BOOL_TO_REAL(xRotatingField);
arMeasurementsGroup2[18] := rTotalReactiveEnergy;
END_ACTION
ACTION actTypConfig:
typConfig_750_495.typChannelConfig[1].xEnableUserScaling:= TRUE;
typConfig_750_495.typChannelConfig[1].wCurrentTransformerRatio :=CurrentRatioPQ1;

typConfig_750_495.typChannelConfig[2].xEnableUserScaling:= TRUE;
typConfig_750_495.typChannelConfig[2].wCurrentTransformerRatio :=CurrentRatioPQ1;

typConfig_750_495.typChannelConfig[3].xEnableUserScaling:= TRUE;
typConfig_750_495.typChannelConfig[3].wCurrentTransformerRatio :=CurrentRatioPQ1;

typConfig_750_495.xWriteConfig := TRUE;
END_ACTION

(* POU 04. Frequency based Bus Select/Group1, FBD *)
PROGRAM Group1
VAR
	Switch1: fbSwitchRelaysBatOrGridBus;
	Group1: CHP_Switch_Handler;
	temp: BOOL;
END_VAR
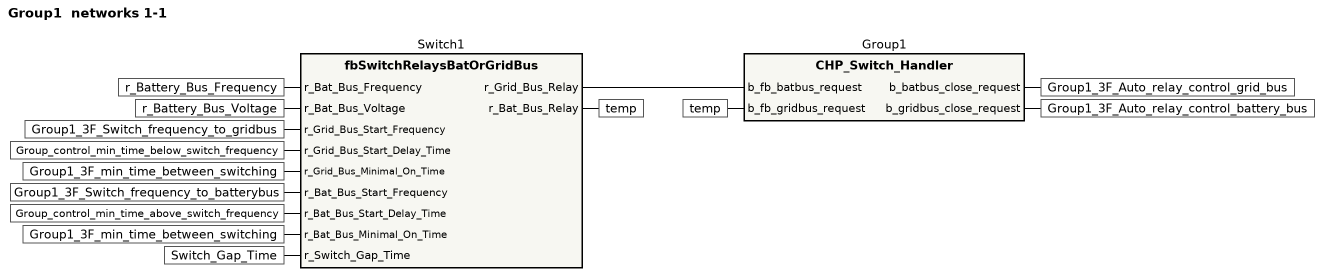
_FBD_ (* Function Block Diagram *)
NETWORK 1
	Group1:CHP_Switch_Handler(b_fb_batbus_request: Switch1:fbSwitchRelaysBatOrGridBus(r_Bat_Bus_Frequency: r_Battery_Bus_Frequency, r_Bat_Bus_Voltage: r_Battery_Bus_Voltage, r_Grid_Bus_Start_Frequency: Group1_3F_Switch_frequency_to_gridbus, r_Grid_Bus_Start_Delay_Time: Group_control_min_time_below_switch_frequency, r_Grid_Bus_Minimal_On_Time: Group1_3F_min_time_between_switching, r_Bat_Bus_Start_Frequency: Group1_3F_Switch_frequency_to_batterybus, r_Bat_Bus_Start_Delay_Time: Group_control_min_time_above_switch_frequency, r_Bat_Bus_Minimal_On_Time: Group1_3F_min_time_between_switching, r_Switch_Gap_Time: Switch_Gap_Time, r_Bat_Bus_Relay => temp), b_fb_gridbus_request: temp, b_gridbus_close_request => Group1_3F_Auto_relay_control_battery_bus) => Group1_3F_Auto_relay_control_grid_bus
_END_FBD_
(* the same logic as Structured Text *)
(* Network 1 *)
Switch1(r_Bat_Bus_Frequency := r_Battery_Bus_Frequency, r_Bat_Bus_Voltage := r_Battery_Bus_Voltage, r_Grid_Bus_Start_Frequency := Group1_3F_Switch_frequency_to_gridbus, r_Grid_Bus_Start_Delay_Time := Group_control_min_time_below_switch_frequency, r_Grid_Bus_Minimal_On_Time := Group1_3F_min_time_between_switching, r_Bat_Bus_Start_Frequency := Group1_3F_Switch_frequency_to_batterybus, r_Bat_Bus_Start_Delay_Time := Group_control_min_time_above_switch_frequency, r_Bat_Bus_Minimal_On_Time := Group1_3F_min_time_between_switching, r_Switch_Gap_Time := Switch_Gap_Time);
temp := Switch1.r_Bat_Bus_Relay;
Group1(b_fb_batbus_request := Switch1.r_Grid_Bus_Relay, b_fb_gridbus_request := temp);
Group1_3F_Auto_relay_control_battery_bus := Group1.b_gridbus_close_request;
Group1_3F_Auto_relay_control_grid_bus := Group1.b_batbus_close_request;
END_PROGRAM

(* POU 04. Frequency based Bus Select/CHP_Switch_Handler, ST *)
FUNCTION_BLOCK CHP_Switch_Handler

VAR_INPUT

	b_fb_batbus_request								:	BOOL; (* request based on frequency, has delayed switching!! *)
	b_fb_gridbus_request							:	BOOL; (* request based on frequency, has delayed switching!! *)

END_VAR

VAR_OUTPUT

	b_batbus_close_request							:	BOOL; (* request based on frequency, has delayed switching!! *)
	b_gridbus_close_request							:	BOOL; (* request based on frequency, has delayed switching!! *)

END_VAR

VAR
(* ____________________________  USED GLOBAL VARIABLES  ___________________________ *)
(*
	(* INPUTS *)
	CHP_control_internal_contacter_switch_state  			AT %IX121.15 : BOOL;
	Group1_3F_Selector_auto_bus_select    				AT %IX121.2 : BOOL;
	Group1_3F_relay_state_battery_bus   					AT %IX120.1  : BOOL;
	Group1_3F_relay_state_grid_bus   						AT %IX120.0  : BOOL;

	(* OUTPUTS *)
	Group1_3F_Auto_relay_control_battery_bus   			AT %QX128.1  : BOOL;
	Group1_3F_Auto_relay_control_grid_bus   				AT %QX128.0  : BOOL;
	CHP_control_Offgrid_request    							AT %QX129.4  : BOOL;
*)
END_VAR
(* CHP handler uses frequency based switching input to control real CHP swithcing when auto input is high *)
(* CHP handler delays switching, such that the CHP can depower and disconnect before switch *)
(* CHP handler delays on-switching, making sure the CHP is disconnected. *)
(* CHP handler delays on-switching, making sure the CHP will connect to the right bus (in the right mode). *)

(* ____________________________  AUTO SWITCH CONTROL  ___________________________ *)
IF Group1_3F_Selector_auto_bus_select THEN
	(*check if wanted state to CHP signal is right, change when required *)
	IF b_fb_gridbus_request THEN
		CHP_control_Offgrid_request :=FALSE;
	ELSE
		IF b_fb_batbus_request THEN
		CHP_control_Offgrid_request :=TRUE;
		END_IF
	END_IF

	(* perform switch between busses when CHP has disconnceted *)
	IF CHP_control_internal_contacter_switch_state = FALSE THEN
		(* Close bat relais when grid relais is open en bat request is still true*)
		IF b_fb_batbus_request THEN
			b_gridbus_close_request := FALSE; (* Disconnect *)
			IF Group1_3F_relay_state_grid_bus = FALSE THEN
				b_batbus_close_request := TRUE;
			END_IF
		END_IF

		(* Close grid relais when bat relais is open en grid request is still true*)
		IF b_fb_gridbus_request THEN
			b_batbus_close_request := FALSE; (* Disconnect *)
			IF Group1_3F_relay_state_battery_bus = FALSE THEN
				b_gridbus_close_request := TRUE;
			END_IF
		END_IF
	END_IF


(* ____________________________  MANUAL CONTROL  ___________________________ *)
ELSE
	(* check if batbus relais is closed, if so, request offgrid (via wanted state *)
	IF Group1_3F_relay_state_battery_bus THEN
		CHP_control_Offgrid_request :=TRUE;
	ELSE (* IF Group1_3F_relay_state_grid_bus THEN *)
		CHP_control_Offgrid_request :=FALSE;
	END_IF
END_IF
END_FUNCTION_BLOCK

(* POU 04. Frequency based Bus Select/temp, ST *)
PROGRAM temp
VAR
	b_DI_Group_AskedState_Grid					:	BOOL; (* NOT jet available !!!!!!!!!!! *)
	b_DI_Group_AskedState_Battery				:	BOOL; (* NOT jet available !!!!!!!!!!! *)
	b_DI_Group_AskedState_Auto					:	BOOL;
	b_DI_CHP_Sync_Contactor						:	BOOL;
	b_batbus_switch_state							:	BOOL;
	b_gridbus_switch_state							:	BOOL;
END_VAR
(* what happens when no automated switching is performed? REQUESTED STATE IS DETERMINED BY RELAIS STATE *)
	IF b_DI_Group_AskedState_Grid THEN
		b_Wanted_state_To_CHP := FALSE;

		(*IF r_BAT_BUS_Grid_Relay THEN*)
			IF  b_DI_CHP_Sync_Contactor = FALSE THEN
				b_Grid_Relay := FALSE;
				b_Bat_Relay := TRUE;
			END_IF
		(*END_IF*)
	ELSE IF b_DI_Group_AskedState_Battery THEN
		(*r_Wanted_state_To_CHP := TRUE;*)

		(*IF r_On_Grid_Relay THEN*)
			IF  b_DI_CHP_Sync_Contactor = FALSE THEN
					b_Bat_Relay := TRUE;
					b_Grid_Relay := FALSE;
			END_IF
		(*END_IF*)
	ELSE
		(* performe swithcing (only when CHP is disconnected) *)
		IF b_Bat_Relay THEN
				IF  b_DI_CHP_Sync_Contactor = FALSE THEN
						b_Bat_Relay := FALSE;
						b_Grid_Relay := TRUE;
				END_IF
		END_IF
		IF b_Grid_Relay THEN
				IF  b_DI_CHP_Sync_Contactor = FALSE THEN
						b_Bat_Relay := TRUE;
						b_Grid_Relay := FALSE;
				END_IF
		END_IF
END_IF
END_IF


(* ____________________________ OLD ___________________________ *)
Group1_gridbus_switch_state := r_Grid_Relay;
Group1_batterybus_switch_state := r_Bat_Relay;

(* parameters *)
Group_control_Frequencybased_bus_selecting_state
r_DI_Group_AskedState_Grid := Group1_autoswitch_state;
r_DI_CHP_Sync_Contactor: = CHP_control_internal_contacter_switch_state;
Group1_autoswitch_state

CHP_gridbus_switch_state 		(* request based on frequency *)
CHP_batterybus_switch_state  	(* request based on frequency *)
END_PROGRAM

(* POU 01. PowerQualityMeasurements/run_PQ, ST *)
PROGRAM run_PQ
VAR
	y: INT;
END_VAR
y:=y+1;
(* gridbus, batbus and connector monitoring *)

PQ_A();									(* postion : 11 *)
	r_Grid_Bus_Frequency			:= 	arMeasurementsGroupA[7];
	r_Grid_Bus_Voltage				:= 	arMeasurementsGroupA[13];

PQ_B();									(* postion : 1 *)
	r_Battery_Bus_Frequency		:= 	arMeasurementsGroupB[7];
	r_Battery_Bus_Voltage			:= 	arMeasurementsGroupB[13];

PQ_Janitza_Battery_Bus();

(* groups monitoring *)
PQ_1();									(* postion : 2 *)
PQ_2();									(* postion : 3 *)
PQ_3();									(* postion : 4 *)
PQ_4();									(* postion : 5 *)
PQ_5();									(* postion : 6 *)
PQ_6();									(* postion : 7 *)
PQ_7();									(* postion : 8 *)
PQ_8();									(* postion : 9 *)
PQ_9();									(* postion : 10 *)
END_PROGRAM

(* POU 01. PowerQualityMeasurements/PQ_A, FBD *)
PROGRAM PQ_A
VAR
	abProcessImageInput	AT %IW120		: ARRAY[0..23] OF BYTE;
	abProcessImageOutput 	AT %QW128		: ARRAY[0..23] OF BYTE;

	bToken										: BYTE;

	State_750_495 							: Fb_750_495_State;
		typ_750_495_State 						: typ_750_495_State;

	Configuration_750_495					: Fb_750_495_Configuration;
		typConfig_750_495						: typConfig_750_495;
		xReadyConfig								: BOOL;
		bFeedbackConfig							: BYTE;

	AC_Compact_01_750_495				: Fb_750_495_AC_Compact_01;
		rTotalActivePower							: REAL;
		rTotalReactivePower						: REAL;
		rTotalApparentPower						: REAL;
		rTotalPowerFactorPF						: REAL;
		rTotalActiveEnergy							: REAL;
		rTotalReactiveEnergy						: REAL;
		rTotalApparentEnergy						: REAL;
		rCurrentN									: REAL;
		xRotatingField								: BOOL;
		arCurrent									: ARRAY[1..3] OF REAL;
		axOvercurrent								: ARRAY[1..3] OF BOOL;
		arVoltage_L_N							: ARRAY[1..3] OF REAL;
		axUndervoltage							: ARRAY[1..3] OF BOOL;
		axOvervoltage								: ARRAY[1..3] OF BOOL;
		arActivePower								: ARRAY[1..3] OF REAL;
		arReactivePower							: ARRAY[1..3] OF REAL;
		arApparentPower							: ARRAY[1..3] OF REAL;
		arCosPhi									: ARRAY[1..3] OF REAL;
		arPowerFactorPF							: ARRAY[1..3] OF REAL;
		arFrequency								: ARRAY[1..3] OF REAL;
		axNoZero									: ARRAY[1..3] OF BOOL;
		axVoltSag									: ARRAY[1..3] OF BOOL;
		ai4Quadrant								: ARRAY[1..3] OF INT;

		xReadyCompact_01						: BOOL;
		abFeedbackCompact_01					: ARRAY[1..8] OF BYTE;


END_VAR
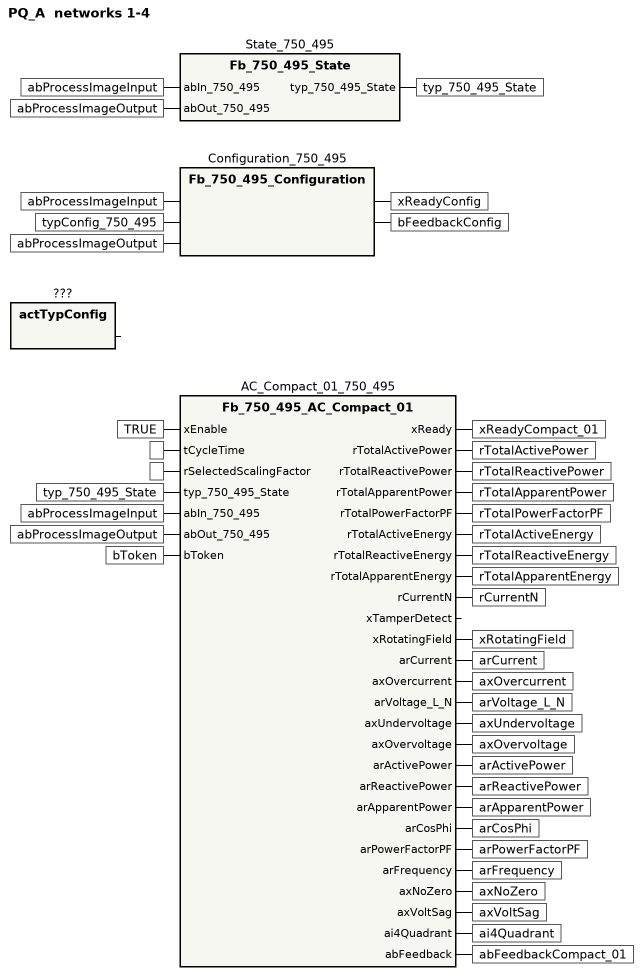
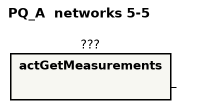
_FBD_ (* Function Block Diagram *)
NETWORK 1
	State_750_495:Fb_750_495_State(abIn_750_495: abProcessImageInput, abOut_750_495: abProcessImageOutput) => typ_750_495_State
NETWORK 2
	Configuration_750_495:Fb_750_495_Configuration(abProcessImageInput, typConfig_750_495, abProcessImageOutput, out 2 => bFeedbackConfig) => xReadyConfig
NETWORK 3
	???:actTypConfig()
NETWORK 4
	AC_Compact_01_750_495:Fb_750_495_AC_Compact_01(xEnable: TRUE, tCycleTime: , rSelectedScalingFactor: , typ_750_495_State: typ_750_495_State, abIn_750_495: abProcessImageInput, abOut_750_495: abProcessImageOutput, bToken: bToken, rTotalActivePower => rTotalActivePower, rTotalReactivePower => rTotalReactivePower, rTotalApparentPower => rTotalApparentPower, rTotalPowerFactorPF => rTotalPowerFactorPF, rTotalActiveEnergy => rTotalActiveEnergy, rTotalReactiveEnergy => rTotalReactiveEnergy, rTotalApparentEnergy => rTotalApparentEnergy, rCurrentN => rCurrentN, xRotatingField => xRotatingField, arCurrent => arCurrent, axOvercurrent => axOvercurrent, arVoltage_L_N => arVoltage_L_N, axUndervoltage => axUndervoltage, axOvervoltage => axOvervoltage, arActivePower => arActivePower, arReactivePower => arReactivePower, arApparentPower => arApparentPower, arCosPhi => arCosPhi, arPowerFactorPF => arPowerFactorPF, arFrequency => arFrequency, axNoZero => axNoZero, axVoltSag => axVoltSag, ai4Quadrant => ai4Quadrant, abFeedback => abFeedbackCompact_01) => xReadyCompact_01
NETWORK 5
	???:actGetMeasurements()
_END_FBD_
(* the same logic as Structured Text *)
(* Network 1 *)
State_750_495(abIn_750_495 := abProcessImageInput, abOut_750_495 := abProcessImageOutput);
typ_750_495_State := State_750_495.typ_750_495_State;
(* Network 2: see the listing above *)
(* Network 3: see the listing above *)
(* Network 4: see the listing above *)
(* Network 5: see the listing above *)
END_PROGRAM
ACTION actGetMeasurements:
arMeasurementsGroupA[1] := arActivePower[1];
arMeasurementsGroupA[2] := arActivePower[2];
arMeasurementsGroupA[3] := arActivePower[3];
arMeasurementsGroupA[4] := arReactivePower[1];
arMeasurementsGroupA[5] := arReactivePower[2];
arMeasurementsGroupA[6] := arReactivePower[3];
arMeasurementsGroupA[7] := arVoltage_L_N[1];
arMeasurementsGroupA[8] := arVoltage_L_N[2];
arMeasurementsGroupA[9] := arVoltage_L_N[3];
arMeasurementsGroupA[10] := arCurrent[1];
arMeasurementsGroupA[11] := arCurrent[2];
arMeasurementsGroupA[12] := arCurrent[3];
arMeasurementsGroupA[13] := arFrequency[1];
arMeasurementsGroupA[14] := arFrequency[2];
arMeasurementsGroupA[15] := arFrequency[3];
arMeasurementsGroupA[16] := rTotalActiveEnergy;
arMeasurementsGroupA[17] := BOOL_TO_REAL(xRotatingField);
arMeasurementsGroupA[18] := rTotalReactiveEnergy;

(* variables used internally, eg auto switching *)
r_Grid_Bus_Frequency := arFrequency[1];
r_Grid_Bus_Voltage := arVoltage_L_N[1];
END_ACTION
ACTION actTypConfig:
typConfig_750_495.typChannelConfig[1].xEnableUserScaling:= TRUE;
typConfig_750_495.typChannelConfig[1].wCurrentTransformerRatio :=CurrentRatioPQ1;

typConfig_750_495.typChannelConfig[2].xEnableUserScaling:= TRUE;
typConfig_750_495.typChannelConfig[2].wCurrentTransformerRatio :=CurrentRatioPQ1;

typConfig_750_495.typChannelConfig[3].xEnableUserScaling:= TRUE;
typConfig_750_495.typChannelConfig[3].wCurrentTransformerRatio :=CurrentRatioPQ1;

typConfig_750_495.xWriteConfig := TRUE;
END_ACTION

(* POU 01. PowerQualityMeasurements/PQ_B, FBD *)
PROGRAM PQ_B
VAR
	abProcessImageInput	AT %IW0			: ARRAY[0..23] OF BYTE;
	abProcessImageOutput 	AT %QW8 			: ARRAY[0..23] OF BYTE;

	bToken										: BYTE;

	State_750_495 							: Fb_750_495_State;
		typ_750_495_State 						: typ_750_495_State;

	Configuration_750_495					: Fb_750_495_Configuration;
		typConfig_750_495						: typConfig_750_495;
		xReadyConfig								: BOOL;
		bFeedbackConfig							: BYTE;

	AC_Compact_01_750_495				: Fb_750_495_AC_Compact_01;
		rTotalActivePower							: REAL;
		rTotalReactivePower						: REAL;
		rTotalApparentPower						: REAL;
		rTotalPowerFactorPF						: REAL;
		rTotalActiveEnergy							: REAL;
		rTotalReactiveEnergy						: REAL;
		rTotalApparentEnergy						: REAL;
		rCurrentN									: REAL;
		xRotatingField								: BOOL;
		arCurrent									: ARRAY[1..3] OF REAL;
		axOvercurrent								: ARRAY[1..3] OF BOOL;
		arVoltage_L_N							: ARRAY[1..3] OF REAL;
		axUndervoltage							: ARRAY[1..3] OF BOOL;
		axOvervoltage								: ARRAY[1..3] OF BOOL;
		arActivePower								: ARRAY[1..3] OF REAL;
		arReactivePower							: ARRAY[1..3] OF REAL;
		arApparentPower							: ARRAY[1..3] OF REAL;
		arCosPhi									: ARRAY[1..3] OF REAL;
		arPowerFactorPF							: ARRAY[1..3] OF REAL;
		arFrequency								: ARRAY[1..3] OF REAL;
		axNoZero									: ARRAY[1..3] OF BOOL;
		axVoltSag									: ARRAY[1..3] OF BOOL;
		ai4Quadrant								: ARRAY[1..3] OF INT;

		xReadyCompact_01						: BOOL;
		abFeedbackCompact_01					: ARRAY[1..8] OF BYTE;


END_VAR
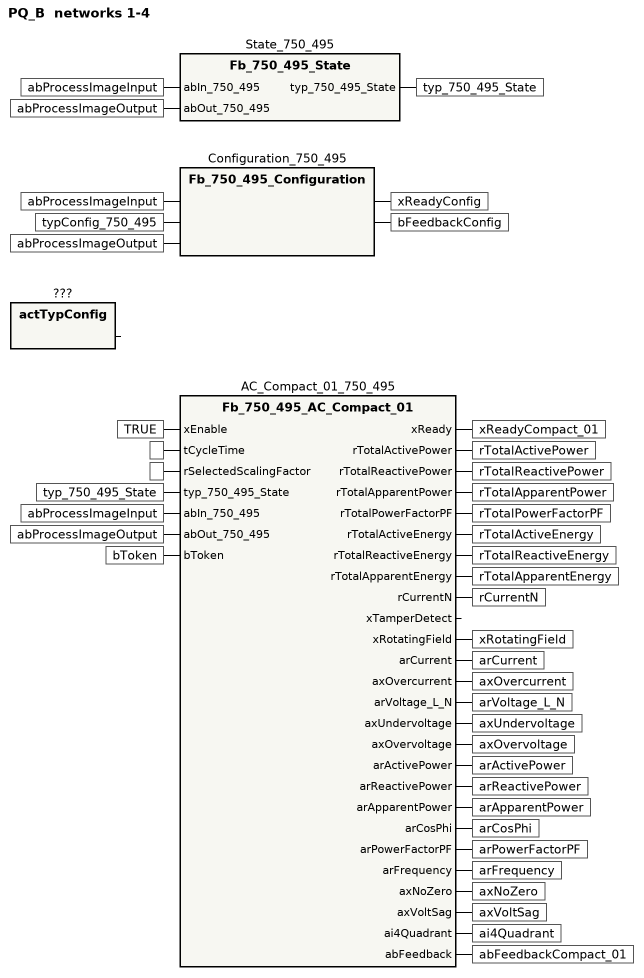
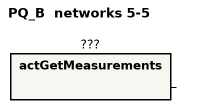
_FBD_ (* Function Block Diagram *)
NETWORK 1
	State_750_495:Fb_750_495_State(abIn_750_495: abProcessImageInput, abOut_750_495: abProcessImageOutput) => typ_750_495_State
NETWORK 2
	Configuration_750_495:Fb_750_495_Configuration(abProcessImageInput, typConfig_750_495, abProcessImageOutput, out 2 => bFeedbackConfig) => xReadyConfig
NETWORK 3
	???:actTypConfig()
NETWORK 4
	AC_Compact_01_750_495:Fb_750_495_AC_Compact_01(xEnable: TRUE, tCycleTime: , rSelectedScalingFactor: , typ_750_495_State: typ_750_495_State, abIn_750_495: abProcessImageInput, abOut_750_495: abProcessImageOutput, bToken: bToken, rTotalActivePower => rTotalActivePower, rTotalReactivePower => rTotalReactivePower, rTotalApparentPower => rTotalApparentPower, rTotalPowerFactorPF => rTotalPowerFactorPF, rTotalActiveEnergy => rTotalActiveEnergy, rTotalReactiveEnergy => rTotalReactiveEnergy, rTotalApparentEnergy => rTotalApparentEnergy, rCurrentN => rCurrentN, xRotatingField => xRotatingField, arCurrent => arCurrent, axOvercurrent => axOvercurrent, arVoltage_L_N => arVoltage_L_N, axUndervoltage => axUndervoltage, axOvervoltage => axOvervoltage, arActivePower => arActivePower, arReactivePower => arReactivePower, arApparentPower => arApparentPower, arCosPhi => arCosPhi, arPowerFactorPF => arPowerFactorPF, arFrequency => arFrequency, axNoZero => axNoZero, axVoltSag => axVoltSag, ai4Quadrant => ai4Quadrant, abFeedback => abFeedbackCompact_01) => xReadyCompact_01
NETWORK 5
	???:actGetMeasurements()
_END_FBD_
(* the same logic as Structured Text *)
(* Network 1 *)
State_750_495(abIn_750_495 := abProcessImageInput, abOut_750_495 := abProcessImageOutput);
typ_750_495_State := State_750_495.typ_750_495_State;
(* Network 2: see the listing above *)
(* Network 3: see the listing above *)
(* Network 4: see the listing above *)
(* Network 5: see the listing above *)
END_PROGRAM
ACTION actGetMeasurements:
arMeasurementsGroupB[1] := arActivePower[1];
arMeasurementsGroupB[2] := arActivePower[2];
arMeasurementsGroupB[3] := arActivePower[3];
arMeasurementsGroupB[4] := arReactivePower[1];
arMeasurementsGroupB[5] := arReactivePower[2];
arMeasurementsGroupB[6] := arReactivePower[3];
arMeasurementsGroupB[7] := arVoltage_L_N[1];
arMeasurementsGroupB[8] := arVoltage_L_N[2];
arMeasurementsGroupB[9] := arVoltage_L_N[3];
arMeasurementsGroupB[10] := arCurrent[1];
arMeasurementsGroupB[11] := arCurrent[2];
arMeasurementsGroupB[12] := arCurrent[3];
arMeasurementsGroupB[13] := arFrequency[1];
arMeasurementsGroupB[14] := arFrequency[2];
arMeasurementsGroupB[15] := arFrequency[3];
arMeasurementsGroupB[16] := rTotalActiveEnergy;
arMeasurementsGroupB[17] := BOOL_TO_REAL(xRotatingField);
arMeasurementsGroupB[18] := rTotalReactiveEnergy;

(* variables used internally, eg auto switching *)
r_Battery_Bus_Frequency := arFrequency[1];
r_Battery_Bus_Voltage := arVoltage_L_N[1];
END_ACTION
ACTION actTypConfig:
typConfig_750_495.typChannelConfig[1].xEnableUserScaling:= TRUE;
typConfig_750_495.typChannelConfig[1].wCurrentTransformerRatio :=CurrentRatioPQ1;

typConfig_750_495.typChannelConfig[2].xEnableUserScaling:= TRUE;
typConfig_750_495.typChannelConfig[2].wCurrentTransformerRatio :=CurrentRatioPQ1;

typConfig_750_495.typChannelConfig[3].xEnableUserScaling:= TRUE;
typConfig_750_495.typChannelConfig[3].wCurrentTransformerRatio :=CurrentRatioPQ1;

typConfig_750_495.xWriteConfig := TRUE;
END_ACTION

(* POU 01. PowerQualityMeasurements/PQ_Janitza_Battery_Bus, ST *)
PROGRAM PQ_Janitza_Battery_Bus
(*  Link to modbus example: https://wiki.janitza.de/display/GRIDVIS70EN/UMG+604+-+Modbus  *)
(* Link to modbus commands/registers:  https://www.janitza.com/manuals.html          UMG 509 Modbus address and formulary (English)  *)
VAR
	y: REAL;
END_VAR
(* to be implemented: arMeasurementsJanitza[x] := Janitza_Modbus[y];*)

y:=y+1; (*TEST*)

(* to be matched from janitza modbus *)

	Bus_Connector_L1_P := y;
END_PROGRAM

(* POU 01. PowerQualityMeasurements/PQ_3, FBD *)
PROGRAM PQ_3
VAR
	abProcessImageInput	AT %IW36			: ARRAY[0..23] OF BYTE;
	abProcessImageOutput 	AT %QW44		: ARRAY[0..23] OF BYTE;

	bToken										: BYTE;

	State_750_495 							: Fb_750_495_State;
		typ_750_495_State 						: typ_750_495_State;

	Configuration_750_495					: Fb_750_495_Configuration;
		typConfig_750_495						: typConfig_750_495;
		xReadyConfig								: BOOL;
		bFeedbackConfig							: BYTE;

	AC_Compact_01_750_495				: Fb_750_495_AC_Compact_01;
		rTotalActivePower							: REAL;
		rTotalReactivePower						: REAL;
		rTotalApparentPower						: REAL;
		rTotalPowerFactorPF						: REAL;
		rTotalActiveEnergy							: REAL;
		rTotalReactiveEnergy						: REAL;
		rTotalApparentEnergy						: REAL;
		rCurrentN									: REAL;
		xRotatingField								: BOOL;
		arCurrent									: ARRAY[1..3] OF REAL;
		axOvercurrent								: ARRAY[1..3] OF BOOL;
		arVoltage_L_N							: ARRAY[1..3] OF REAL;
		axUndervoltage							: ARRAY[1..3] OF BOOL;
		axOvervoltage								: ARRAY[1..3] OF BOOL;
		arActivePower								: ARRAY[1..3] OF REAL;
		arReactivePower							: ARRAY[1..3] OF REAL;
		arApparentPower							: ARRAY[1..3] OF REAL;
		arCosPhi									: ARRAY[1..3] OF REAL;
		arPowerFactorPF							: ARRAY[1..3] OF REAL;
		arFrequency								: ARRAY[1..3] OF REAL;
		axNoZero									: ARRAY[1..3] OF BOOL;
		axVoltSag									: ARRAY[1..3] OF BOOL;
		ai4Quadrant								: ARRAY[1..3] OF INT;

		xReadyCompact_01						: BOOL;
		abFeedbackCompact_01					: ARRAY[1..8] OF BYTE;


END_VAR
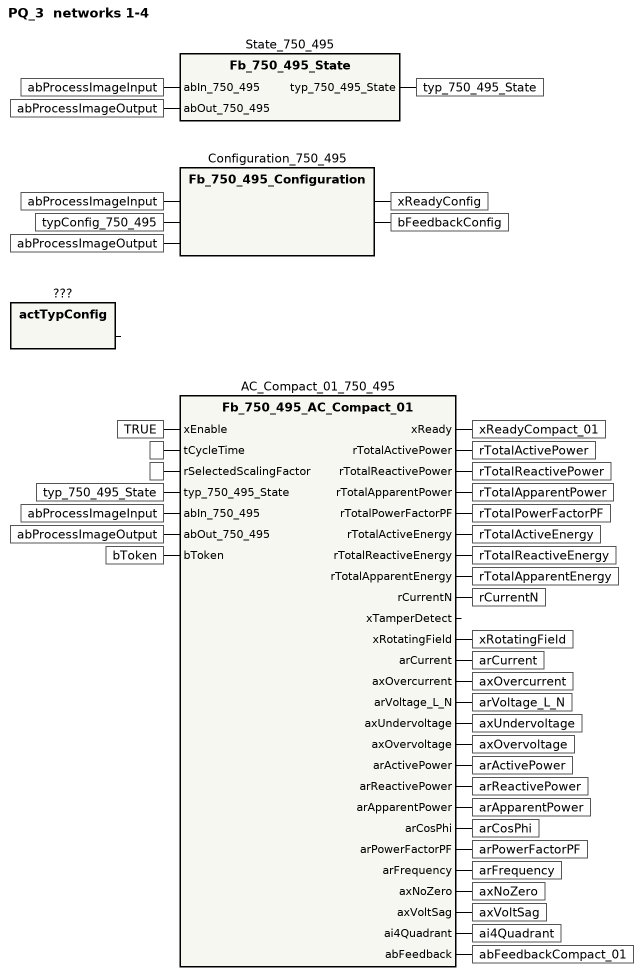
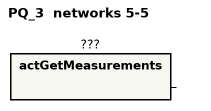
_FBD_ (* Function Block Diagram *)
NETWORK 1
	State_750_495:Fb_750_495_State(abIn_750_495: abProcessImageInput, abOut_750_495: abProcessImageOutput) => typ_750_495_State
NETWORK 2
	Configuration_750_495:Fb_750_495_Configuration(abProcessImageInput, typConfig_750_495, abProcessImageOutput, out 2 => bFeedbackConfig) => xReadyConfig
NETWORK 3
	???:actTypConfig()
NETWORK 4
	AC_Compact_01_750_495:Fb_750_495_AC_Compact_01(xEnable: TRUE, tCycleTime: , rSelectedScalingFactor: , typ_750_495_State: typ_750_495_State, abIn_750_495: abProcessImageInput, abOut_750_495: abProcessImageOutput, bToken: bToken, rTotalActivePower => rTotalActivePower, rTotalReactivePower => rTotalReactivePower, rTotalApparentPower => rTotalApparentPower, rTotalPowerFactorPF => rTotalPowerFactorPF, rTotalActiveEnergy => rTotalActiveEnergy, rTotalReactiveEnergy => rTotalReactiveEnergy, rTotalApparentEnergy => rTotalApparentEnergy, rCurrentN => rCurrentN, xRotatingField => xRotatingField, arCurrent => arCurrent, axOvercurrent => axOvercurrent, arVoltage_L_N => arVoltage_L_N, axUndervoltage => axUndervoltage, axOvervoltage => axOvervoltage, arActivePower => arActivePower, arReactivePower => arReactivePower, arApparentPower => arApparentPower, arCosPhi => arCosPhi, arPowerFactorPF => arPowerFactorPF, arFrequency => arFrequency, axNoZero => axNoZero, axVoltSag => axVoltSag, ai4Quadrant => ai4Quadrant, abFeedback => abFeedbackCompact_01) => xReadyCompact_01
NETWORK 5
	???:actGetMeasurements()
_END_FBD_
(* the same logic as Structured Text *)
(* Network 1 *)
State_750_495(abIn_750_495 := abProcessImageInput, abOut_750_495 := abProcessImageOutput);
typ_750_495_State := State_750_495.typ_750_495_State;
(* Network 2: see the listing above *)
(* Network 3: see the listing above *)
(* Network 4: see the listing above *)
(* Network 5: see the listing above *)
END_PROGRAM
ACTION actGetMeasurements:
arMeasurementsGroup3[1] := arActivePower[1];
arMeasurementsGroup3[2] := arActivePower[2];
arMeasurementsGroup3[3] := arActivePower[3];
arMeasurementsGroup3[4] := arReactivePower[1];
arMeasurementsGroup3[5] := arReactivePower[2];
arMeasurementsGroup3[6] := arReactivePower[3];
arMeasurementsGroup3[7] := arVoltage_L_N[1];
arMeasurementsGroup3[8] := arVoltage_L_N[2];
arMeasurementsGroup3[9] := arVoltage_L_N[3];
arMeasurementsGroup3[10] := arCurrent[1];
arMeasurementsGroup3[11] := arCurrent[2];
arMeasurementsGroup3[12] := arCurrent[3];
arMeasurementsGroup3[13] := arFrequency[1];
arMeasurementsGroup3[14] := arFrequency[2];
arMeasurementsGroup3[15] := arFrequency[3];
arMeasurementsGroup3[16] := rTotalActiveEnergy;
arMeasurementsGroup3[17] := BOOL_TO_REAL(xRotatingField);
arMeasurementsGroup3[18] := rTotalReactiveEnergy;
END_ACTION
ACTION actTypConfig:
typConfig_750_495.typChannelConfig[1].xEnableUserScaling:= TRUE;
typConfig_750_495.typChannelConfig[1].wCurrentTransformerRatio :=CurrentRatioPQ1;

typConfig_750_495.typChannelConfig[2].xEnableUserScaling:= TRUE;
typConfig_750_495.typChannelConfig[2].wCurrentTransformerRatio :=CurrentRatioPQ1;

typConfig_750_495.typChannelConfig[3].xEnableUserScaling:= TRUE;
typConfig_750_495.typChannelConfig[3].wCurrentTransformerRatio :=CurrentRatioPQ1;

typConfig_750_495.xWriteConfig := TRUE;
END_ACTION

(* POU 01. PowerQualityMeasurements/PQ_4, FBD *)
PROGRAM PQ_4
VAR
	abProcessImageInput	AT %IW48			: ARRAY[0..23] OF BYTE;
	abProcessImageOutput 	AT %QW56		: ARRAY[0..23] OF BYTE;

	bToken										: BYTE;

	State_750_495 							: Fb_750_495_State;
		typ_750_495_State 						: typ_750_495_State;

	Configuration_750_495					: Fb_750_495_Configuration;
		typConfig_750_495						: typConfig_750_495;
		xReadyConfig								: BOOL;
		bFeedbackConfig							: BYTE;

	AC_Compact_01_750_495				: Fb_750_495_AC_Compact_01;
		rTotalActivePower							: REAL;
		rTotalReactivePower						: REAL;
		rTotalApparentPower						: REAL;
		rTotalPowerFactorPF						: REAL;
		rTotalActiveEnergy							: REAL;
		rTotalReactiveEnergy						: REAL;
		rTotalApparentEnergy						: REAL;
		rCurrentN									: REAL;
		xRotatingField								: BOOL;
		arCurrent									: ARRAY[1..3] OF REAL;
		axOvercurrent								: ARRAY[1..3] OF BOOL;
		arVoltage_L_N							: ARRAY[1..3] OF REAL;
		axUndervoltage							: ARRAY[1..3] OF BOOL;
		axOvervoltage								: ARRAY[1..3] OF BOOL;
		arActivePower								: ARRAY[1..3] OF REAL;
		arReactivePower							: ARRAY[1..3] OF REAL;
		arApparentPower							: ARRAY[1..3] OF REAL;
		arCosPhi									: ARRAY[1..3] OF REAL;
		arPowerFactorPF							: ARRAY[1..3] OF REAL;
		arFrequency								: ARRAY[1..3] OF REAL;
		axNoZero									: ARRAY[1..3] OF BOOL;
		axVoltSag									: ARRAY[1..3] OF BOOL;
		ai4Quadrant								: ARRAY[1..3] OF INT;

		xReadyCompact_01						: BOOL;
		abFeedbackCompact_01					: ARRAY[1..8] OF BYTE;


END_VAR
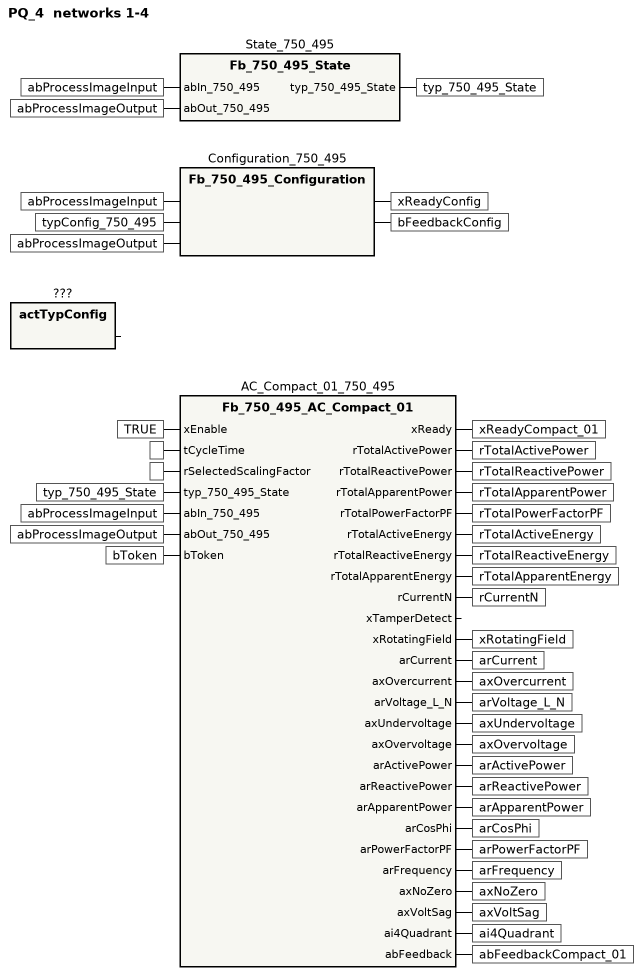
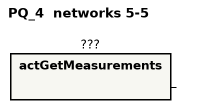
_FBD_ (* Function Block Diagram *)
NETWORK 1
	State_750_495:Fb_750_495_State(abIn_750_495: abProcessImageInput, abOut_750_495: abProcessImageOutput) => typ_750_495_State
NETWORK 2
	Configuration_750_495:Fb_750_495_Configuration(abProcessImageInput, typConfig_750_495, abProcessImageOutput, out 2 => bFeedbackConfig) => xReadyConfig
NETWORK 3
	???:actTypConfig()
NETWORK 4
	AC_Compact_01_750_495:Fb_750_495_AC_Compact_01(xEnable: TRUE, tCycleTime: , rSelectedScalingFactor: , typ_750_495_State: typ_750_495_State, abIn_750_495: abProcessImageInput, abOut_750_495: abProcessImageOutput, bToken: bToken, rTotalActivePower => rTotalActivePower, rTotalReactivePower => rTotalReactivePower, rTotalApparentPower => rTotalApparentPower, rTotalPowerFactorPF => rTotalPowerFactorPF, rTotalActiveEnergy => rTotalActiveEnergy, rTotalReactiveEnergy => rTotalReactiveEnergy, rTotalApparentEnergy => rTotalApparentEnergy, rCurrentN => rCurrentN, xRotatingField => xRotatingField, arCurrent => arCurrent, axOvercurrent => axOvercurrent, arVoltage_L_N => arVoltage_L_N, axUndervoltage => axUndervoltage, axOvervoltage => axOvervoltage, arActivePower => arActivePower, arReactivePower => arReactivePower, arApparentPower => arApparentPower, arCosPhi => arCosPhi, arPowerFactorPF => arPowerFactorPF, arFrequency => arFrequency, axNoZero => axNoZero, axVoltSag => axVoltSag, ai4Quadrant => ai4Quadrant, abFeedback => abFeedbackCompact_01) => xReadyCompact_01
NETWORK 5
	???:actGetMeasurements()
_END_FBD_
(* the same logic as Structured Text *)
(* Network 1 *)
State_750_495(abIn_750_495 := abProcessImageInput, abOut_750_495 := abProcessImageOutput);
typ_750_495_State := State_750_495.typ_750_495_State;
(* Network 2: see the listing above *)
(* Network 3: see the listing above *)
(* Network 4: see the listing above *)
(* Network 5: see the listing above *)
END_PROGRAM
ACTION actGetMeasurements:
arMeasurementsGroup4[1] := arActivePower[1];
arMeasurementsGroup4[2] := arActivePower[2];
arMeasurementsGroup4[3] := arActivePower[3];
arMeasurementsGroup4[4] := arReactivePower[1];
arMeasurementsGroup4[5] := arReactivePower[2];
arMeasurementsGroup4[6] := arReactivePower[3];
arMeasurementsGroup4[7] := arVoltage_L_N[1];
arMeasurementsGroup4[8] := arVoltage_L_N[2];
arMeasurementsGroup4[9] := arVoltage_L_N[3];
arMeasurementsGroup4[10] := arCurrent[1];
arMeasurementsGroup4[11] := arCurrent[2];
arMeasurementsGroup4[12] := arCurrent[3];
arMeasurementsGroup4[13] := arFrequency[1];
arMeasurementsGroup4[14] := arFrequency[2];
arMeasurementsGroup4[15] := arFrequency[3];
arMeasurementsGroup4[16] := rTotalActiveEnergy;
arMeasurementsGroup4[17] := BOOL_TO_REAL(xRotatingField);
arMeasurementsGroup4[18] := rTotalReactiveEnergy;
END_ACTION
ACTION actTypConfig:
typConfig_750_495.typChannelConfig[1].xEnableUserScaling:= TRUE;
typConfig_750_495.typChannelConfig[1].wCurrentTransformerRatio :=CurrentRatioPQ1;

typConfig_750_495.typChannelConfig[2].xEnableUserScaling:= TRUE;
typConfig_750_495.typChannelConfig[2].wCurrentTransformerRatio :=CurrentRatioPQ1;

typConfig_750_495.typChannelConfig[3].xEnableUserScaling:= TRUE;
typConfig_750_495.typChannelConfig[3].wCurrentTransformerRatio :=CurrentRatioPQ1;

typConfig_750_495.xWriteConfig := TRUE;
END_ACTION

(* POU 01. PowerQualityMeasurements/PQ_5, FBD *)
PROGRAM PQ_5
VAR
	abProcessImageInput	AT %IW60			: ARRAY[0..23] OF BYTE;
	abProcessImageOutput 	AT %QW68		: ARRAY[0..23] OF BYTE;

	bToken										: BYTE;

	State_750_495 							: Fb_750_495_State;
		typ_750_495_State 						: typ_750_495_State;

	Configuration_750_495					: Fb_750_495_Configuration;
		typConfig_750_495						: typConfig_750_495;
		xReadyConfig								: BOOL;
		bFeedbackConfig							: BYTE;

	AC_Compact_01_750_495				: Fb_750_495_AC_Compact_01;
		rTotalActivePower							: REAL;
		rTotalReactivePower						: REAL;
		rTotalApparentPower						: REAL;
		rTotalPowerFactorPF						: REAL;
		rTotalActiveEnergy							: REAL;
		rTotalReactiveEnergy						: REAL;
		rTotalApparentEnergy						: REAL;
		rCurrentN									: REAL;
		xRotatingField								: BOOL;
		arCurrent									: ARRAY[1..3] OF REAL;
		axOvercurrent								: ARRAY[1..3] OF BOOL;
		arVoltage_L_N							: ARRAY[1..3] OF REAL;
		axUndervoltage							: ARRAY[1..3] OF BOOL;
		axOvervoltage								: ARRAY[1..3] OF BOOL;
		arActivePower								: ARRAY[1..3] OF REAL;
		arReactivePower							: ARRAY[1..3] OF REAL;
		arApparentPower							: ARRAY[1..3] OF REAL;
		arCosPhi									: ARRAY[1..3] OF REAL;
		arPowerFactorPF							: ARRAY[1..3] OF REAL;
		arFrequency								: ARRAY[1..3] OF REAL;
		axNoZero									: ARRAY[1..3] OF BOOL;
		axVoltSag									: ARRAY[1..3] OF BOOL;
		ai4Quadrant								: ARRAY[1..3] OF INT;

		xReadyCompact_01						: BOOL;
		abFeedbackCompact_01					: ARRAY[1..8] OF BYTE;


END_VAR
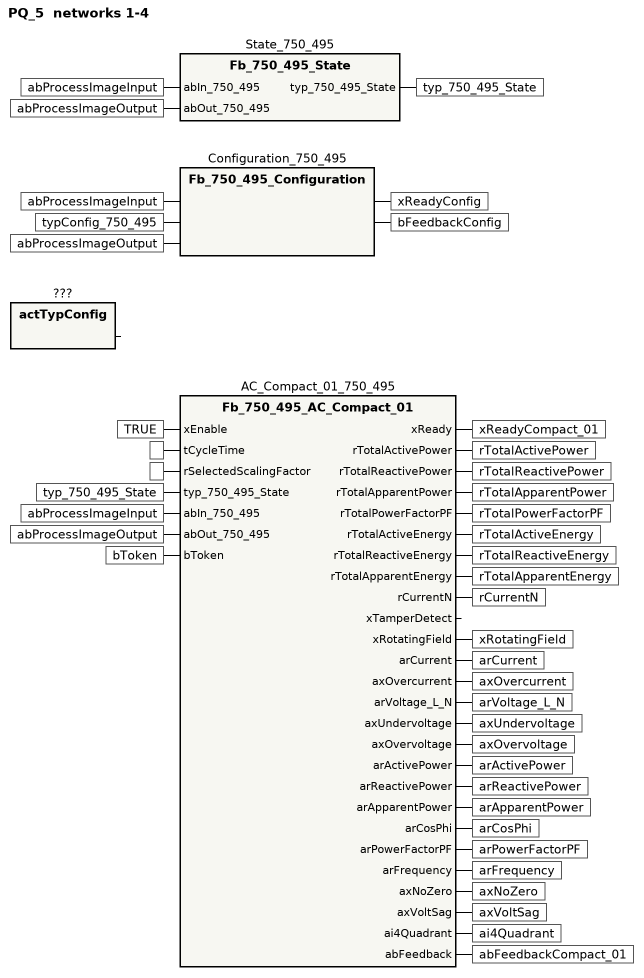
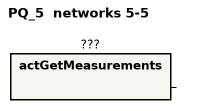
_FBD_ (* Function Block Diagram *)
NETWORK 1
	State_750_495:Fb_750_495_State(abIn_750_495: abProcessImageInput, abOut_750_495: abProcessImageOutput) => typ_750_495_State
NETWORK 2
	Configuration_750_495:Fb_750_495_Configuration(abProcessImageInput, typConfig_750_495, abProcessImageOutput, out 2 => bFeedbackConfig) => xReadyConfig
NETWORK 3
	???:actTypConfig()
NETWORK 4
	AC_Compact_01_750_495:Fb_750_495_AC_Compact_01(xEnable: TRUE, tCycleTime: , rSelectedScalingFactor: , typ_750_495_State: typ_750_495_State, abIn_750_495: abProcessImageInput, abOut_750_495: abProcessImageOutput, bToken: bToken, rTotalActivePower => rTotalActivePower, rTotalReactivePower => rTotalReactivePower, rTotalApparentPower => rTotalApparentPower, rTotalPowerFactorPF => rTotalPowerFactorPF, rTotalActiveEnergy => rTotalActiveEnergy, rTotalReactiveEnergy => rTotalReactiveEnergy, rTotalApparentEnergy => rTotalApparentEnergy, rCurrentN => rCurrentN, xRotatingField => xRotatingField, arCurrent => arCurrent, axOvercurrent => axOvercurrent, arVoltage_L_N => arVoltage_L_N, axUndervoltage => axUndervoltage, axOvervoltage => axOvervoltage, arActivePower => arActivePower, arReactivePower => arReactivePower, arApparentPower => arApparentPower, arCosPhi => arCosPhi, arPowerFactorPF => arPowerFactorPF, arFrequency => arFrequency, axNoZero => axNoZero, axVoltSag => axVoltSag, ai4Quadrant => ai4Quadrant, abFeedback => abFeedbackCompact_01) => xReadyCompact_01
NETWORK 5
	???:actGetMeasurements()
_END_FBD_
(* the same logic as Structured Text *)
(* Network 1 *)
State_750_495(abIn_750_495 := abProcessImageInput, abOut_750_495 := abProcessImageOutput);
typ_750_495_State := State_750_495.typ_750_495_State;
(* Network 2: see the listing above *)
(* Network 3: see the listing above *)
(* Network 4: see the listing above *)
(* Network 5: see the listing above *)
END_PROGRAM
ACTION actGetMeasurements:
arMeasurementsGroup5[1] := arActivePower[1];
arMeasurementsGroup5[2] := arActivePower[2];
arMeasurementsGroup5[3] := arActivePower[3];
arMeasurementsGroup5[4] := arReactivePower[1];
arMeasurementsGroup5[5] := arReactivePower[2];
arMeasurementsGroup5[6] := arReactivePower[3];
arMeasurementsGroup5[7] := arVoltage_L_N[1];
arMeasurementsGroup5[8] := arVoltage_L_N[2];
arMeasurementsGroup5[9] := arVoltage_L_N[3];
arMeasurementsGroup5[10] := arCurrent[1];
arMeasurementsGroup5[11] := arCurrent[2];
arMeasurementsGroup5[12] := arCurrent[3];
arMeasurementsGroup5[13] := arFrequency[1];
arMeasurementsGroup5[14] := arFrequency[2];
arMeasurementsGroup5[15] := arFrequency[3];
arMeasurementsGroup5[16] := rTotalActiveEnergy;
arMeasurementsGroup5[17] := BOOL_TO_REAL(xRotatingField);
arMeasurementsGroup5[18] := rTotalReactiveEnergy;
END_ACTION
ACTION actTypConfig:
typConfig_750_495.typChannelConfig[1].xEnableUserScaling:= TRUE;
typConfig_750_495.typChannelConfig[1].wCurrentTransformerRatio :=CurrentRatioPQ1;

typConfig_750_495.typChannelConfig[2].xEnableUserScaling:= TRUE;
typConfig_750_495.typChannelConfig[2].wCurrentTransformerRatio :=CurrentRatioPQ1;

typConfig_750_495.typChannelConfig[3].xEnableUserScaling:= TRUE;
typConfig_750_495.typChannelConfig[3].wCurrentTransformerRatio :=CurrentRatioPQ1;

typConfig_750_495.xWriteConfig := TRUE;
END_ACTION

(* POU 01. PowerQualityMeasurements/PQ_6, FBD *)
PROGRAM PQ_6
VAR
	abProcessImageInput	AT %IW72			: ARRAY[0..23] OF BYTE;
	abProcessImageOutput 	AT %QW80		: ARRAY[0..23] OF BYTE;

	bToken										: BYTE;

	State_750_495 							: Fb_750_495_State;
		typ_750_495_State 						: typ_750_495_State;

	Configuration_750_495					: Fb_750_495_Configuration;
		typConfig_750_495						: typConfig_750_495;
		xReadyConfig								: BOOL;
		bFeedbackConfig							: BYTE;

	AC_Compact_01_750_495				: Fb_750_495_AC_Compact_01;
		rTotalActivePower							: REAL;
		rTotalReactivePower						: REAL;
		rTotalApparentPower						: REAL;
		rTotalPowerFactorPF						: REAL;
		rTotalActiveEnergy							: REAL;
		rTotalReactiveEnergy						: REAL;
		rTotalApparentEnergy						: REAL;
		rCurrentN									: REAL;
		xRotatingField								: BOOL;
		arCurrent									: ARRAY[1..3] OF REAL;
		axOvercurrent								: ARRAY[1..3] OF BOOL;
		arVoltage_L_N							: ARRAY[1..3] OF REAL;
		axUndervoltage							: ARRAY[1..3] OF BOOL;
		axOvervoltage								: ARRAY[1..3] OF BOOL;
		arActivePower								: ARRAY[1..3] OF REAL;
		arReactivePower							: ARRAY[1..3] OF REAL;
		arApparentPower							: ARRAY[1..3] OF REAL;
		arCosPhi									: ARRAY[1..3] OF REAL;
		arPowerFactorPF							: ARRAY[1..3] OF REAL;
		arFrequency								: ARRAY[1..3] OF REAL;
		axNoZero									: ARRAY[1..3] OF BOOL;
		axVoltSag									: ARRAY[1..3] OF BOOL;
		ai4Quadrant								: ARRAY[1..3] OF INT;

		xReadyCompact_01						: BOOL;
		abFeedbackCompact_01					: ARRAY[1..8] OF BYTE;


END_VAR
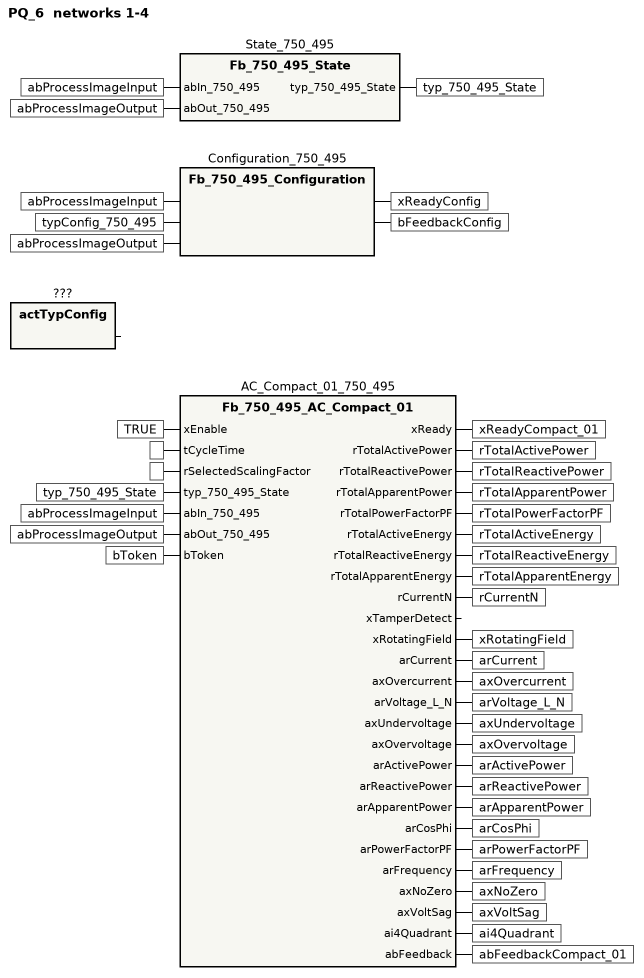
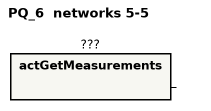
_FBD_ (* Function Block Diagram *)
NETWORK 1
	State_750_495:Fb_750_495_State(abIn_750_495: abProcessImageInput, abOut_750_495: abProcessImageOutput) => typ_750_495_State
NETWORK 2
	Configuration_750_495:Fb_750_495_Configuration(abProcessImageInput, typConfig_750_495, abProcessImageOutput, out 2 => bFeedbackConfig) => xReadyConfig
NETWORK 3
	???:actTypConfig()
NETWORK 4
	AC_Compact_01_750_495:Fb_750_495_AC_Compact_01(xEnable: TRUE, tCycleTime: , rSelectedScalingFactor: , typ_750_495_State: typ_750_495_State, abIn_750_495: abProcessImageInput, abOut_750_495: abProcessImageOutput, bToken: bToken, rTotalActivePower => rTotalActivePower, rTotalReactivePower => rTotalReactivePower, rTotalApparentPower => rTotalApparentPower, rTotalPowerFactorPF => rTotalPowerFactorPF, rTotalActiveEnergy => rTotalActiveEnergy, rTotalReactiveEnergy => rTotalReactiveEnergy, rTotalApparentEnergy => rTotalApparentEnergy, rCurrentN => rCurrentN, xRotatingField => xRotatingField, arCurrent => arCurrent, axOvercurrent => axOvercurrent, arVoltage_L_N => arVoltage_L_N, axUndervoltage => axUndervoltage, axOvervoltage => axOvervoltage, arActivePower => arActivePower, arReactivePower => arReactivePower, arApparentPower => arApparentPower, arCosPhi => arCosPhi, arPowerFactorPF => arPowerFactorPF, arFrequency => arFrequency, axNoZero => axNoZero, axVoltSag => axVoltSag, ai4Quadrant => ai4Quadrant, abFeedback => abFeedbackCompact_01) => xReadyCompact_01
NETWORK 5
	???:actGetMeasurements()
_END_FBD_
(* the same logic as Structured Text *)
(* Network 1 *)
State_750_495(abIn_750_495 := abProcessImageInput, abOut_750_495 := abProcessImageOutput);
typ_750_495_State := State_750_495.typ_750_495_State;
(* Network 2: see the listing above *)
(* Network 3: see the listing above *)
(* Network 4: see the listing above *)
(* Network 5: see the listing above *)
END_PROGRAM
ACTION actGetMeasurements:
arMeasurementsGroup6[1] := arActivePower[1];
arMeasurementsGroup6[2] := arActivePower[2];
arMeasurementsGroup6[3] := arActivePower[3];
arMeasurementsGroup6[4] := arReactivePower[1];
arMeasurementsGroup6[5] := arReactivePower[2];
arMeasurementsGroup6[6] := arReactivePower[3];
arMeasurementsGroup6[7] := arVoltage_L_N[1];
arMeasurementsGroup6[8] := arVoltage_L_N[2];
arMeasurementsGroup6[9] := arVoltage_L_N[3];
arMeasurementsGroup6[10] := arCurrent[1];
arMeasurementsGroup6[11] := arCurrent[2];
arMeasurementsGroup6[12] := arCurrent[3];
arMeasurementsGroup6[13] := arFrequency[1];
arMeasurementsGroup6[14] := arFrequency[2];
arMeasurementsGroup6[15] := arFrequency[3];
arMeasurementsGroup6[16] := rTotalActiveEnergy;
arMeasurementsGroup6[17] := BOOL_TO_REAL(xRotatingField);
arMeasurementsGroup6[18] := rTotalReactiveEnergy;
END_ACTION
ACTION actTypConfig:
typConfig_750_495.typChannelConfig[1].xEnableUserScaling:= TRUE;
typConfig_750_495.typChannelConfig[1].wCurrentTransformerRatio :=CurrentRatioPQ1;

typConfig_750_495.typChannelConfig[2].xEnableUserScaling:= TRUE;
typConfig_750_495.typChannelConfig[2].wCurrentTransformerRatio :=CurrentRatioPQ1;

typConfig_750_495.typChannelConfig[3].xEnableUserScaling:= TRUE;
typConfig_750_495.typChannelConfig[3].wCurrentTransformerRatio :=CurrentRatioPQ1;

typConfig_750_495.xWriteConfig := TRUE;
END_ACTION

(* POU 01. PowerQualityMeasurements/PQ_7, FBD *)
PROGRAM PQ_7
VAR
	abProcessImageInput	AT %IW84			: ARRAY[0..23] OF BYTE;
	abProcessImageOutput 	AT %QW92 			: ARRAY[0..23] OF BYTE;

	bToken										: BYTE;

	State_750_495 							: Fb_750_495_State;
		typ_750_495_State 						: typ_750_495_State;

	Configuration_750_495					: Fb_750_495_Configuration;
		typConfig_750_495						: typConfig_750_495;
		xReadyConfig								: BOOL;
		bFeedbackConfig							: BYTE;

